LIN {X 0,Y 573.722,Z 200.489,A -85,B 0,C 180,E1 -2273.526,E2 -2273.526} C_VEL
LIN {X 0,Y 573.235,Z 198.084,A -85,B 0,C 180,E1 -2273.91,E2 -2273.91} C_VEL
LIN {X 0,Y 573.224,Z 198.082,A -85,B 0,C 180,E1 -2276.489,E2 -2276.489} C_VEL
LIN {X 0,Y 573.223,Z 198.08,A -85,B 0,C 180,E1 -2278.562,E2 -2278.562} C_VEL
LIN {X 0,Y 573.214,Z 198.078,A -85,B 0,C 180,E1 -2280.99,E2 -2280.99} C_VEL
LIN {X 0,Y 573.246,Z 198.076,A -85,B 0,C 180,E1 -2283.521,E2 -2283.521} C_VEL
LIN {X 0,Y 573.237,Z 198.083,A -85,B 0,C 180,E1 -2286.045,E2 -2286.045} C_VEL
LIN {X 0,Y 573.225,Z 198.076,A -85,B 0,C 180,E1 -2288.698,E2 -2288.698} C_VEL
LIN {X 0,Y 573.228,Z 198.081,A -85,B 0,C 180,E1 -2291.592,E2 -2291.592} C_VEL
LIN {X 0,Y 573.21,Z 198.08,A -85,B 0,C 180,E1 -2294.33,E2 -2294.33} C_VEL
LIN {X 0,Y 573.227,Z 198.079,A -85,B 0,C 180,E1 -2297.353,E2 -2297.353} C_VEL
LIN {X 0,Y 573.207,Z 198.079,A -85,B 0,C 180,E1 -2300.389,E2 -2300.389} C_VEL
LIN {X 0,Y 573.218,Z 198.079,A -85,B 0,C 180,E1 -2303.075,E2 -2303.075} C_VEL
LIN {X 0,Y 573.236,Z 198.083,A -85,B 0,C 180,E1 -2305.669,E2 -2305.669} C_VEL
LIN {X 0,Y 573.211,Z 198.079,A -85,B 0,C 180,E1 -2308.182,E2 -2308.182} C_VEL
LIN {X 0,Y 573.224,Z 198.076,A -85,B 0,C 180,E1 -2310.632,E2 -2310.632} C_VEL
LIN {X 0,Y 573.222,Z 198.086,A -85,B 0,C 180,E1 -2313.498,E2 -2313.498} C_VEL
LIN {X 0,Y 573.194,Z 198.08,A -85,B 0,C 180,E1 -2316.133,E2 -2316.133} C_VEL
LIN {X 0,Y 573.208,Z 198.079,A -85,B 0,C 180,E1 -2318.704,E2 -2318.704} C_VEL
LIN {X 0,Y 573.199,Z 198.087,A -85,B 0,C 180,E1 -2321.41,E2 -2321.41} C_VEL
LIN {X 0,Y 573.216,Z 198.081,A -85,B 0,C 180,E1 -2323.62,E2 -2323.62} C_VEL
LIN {X 0,Y 573.186,Z 198.082,A -85,B 0,C 180,E1 -2326.528,E2 -2326.528} C_VEL
LIN {X 0,Y 573.241,Z 198.079,A -85,B 0,C 180,E1 -2329.403,E2 -2329.403} C_VEL
LIN {X 0,Y 573.231,Z 198.075,A -85,B 0,C 180,E1 -2332.249,E2 -2332.249} C_VEL
LIN {X 0,Y 573.262,Z 198.081,A -85,B 0,C 180,E1 -2335.077,E2 -2335.077} C_VEL
LIN {X 0,Y 573.244,Z 198.074,A -85,B 0,C 180,E1 -2337.892,E2 -2337.892} C_VEL
LIN {X 0,Y 573.291,Z 198.074,A -85,B 0,C 180,E1 -2340.702,E2 -2340.702} C_VEL
LIN {X 0,Y 573.194,Z 198.081,A -85,B 0,C 180,E1 -2343.514,E2 -2343.514} C_VEL
LIN {X 0,Y 573.244,Z 198.074,A -85,B 0,C 180,E1 -2345.628,E2 -2345.628} C_VEL
LIN {X 0,Y 573.234,Z 198.075,A -85,B 0,C 180,E1 -2347.75,E2 -2347.75} C_VEL
LIN {X 0,Y 573.247,Z 198.081,A -85,B 0,C 180,E1 -2350.597,E2 -2350.597} C_VEL
LIN {X 0,Y 573.204,Z 198.079,A -85,B 0,C 180,E1 -2353.471,E2 -2353.471} C_VEL
LIN {X 0,Y 573.221,Z 198.082,A -85,B 0,C 180,E1 -2356.379,E2 -2356.379} C_VEL
LIN {X 0,Y 573.222,Z 198.077,A -85,B 0,C 180,E1 -2359.331,E2 -2359.331} C_VEL
LIN {X 0,Y 573.241,Z 198.081,A -85,B 0,C 180,E1 -2362.337,E2 -2362.337} C_VEL
LIN {X 0,Y 573.214,Z 198.082,A -85,B 0,C 180,E1 -2364.433,E2 -2364.433} C_VEL
LIN {X 0,Y 572.574,Z 198.165,A -85,B 0,C 180,E1 -2365.019,E2 -2365.019} C_VEL
LIN {X 0,Y 569.731,Z 198.517,A -85,B 0,C 180,E1 -2365.971,E2 -2365.971} C_VEL
LIN {X 0,Y 567.309,Z 198.818,A -85,B 0,C 180,E1 -2366.737,E2 -2366.737} C_VEL
LIN {X 0,Y 566.26,Z 198.944,A -85,B 0,C 180,E1 -2367.329,E2 -2367.329} C_VEL
LIN {X 0,Y 566.171,Z 198.955,A -85,B 0,C 180,E1 -2367.529,E2 -2367.529} C_VEL
LIN {X 0,Y 566.186,Z 198.954,A -85,B 0,C 180,E1 -2369.769,E2 -2369.769} C_VEL
LIN {X 0,Y 566.172,Z 198.962,A -85,B 0,C 180,E1 -2372.435,E2 -2372.435} C_VEL
LIN {X 0,Y 566.175,Z 198.955,A -85,B 0,C 180,E1 -2374.998,E2 -2374.998} C_VEL
LIN {X 0,Y 566.158,Z 198.957,A -85,B 0,C 180,E1 -2377.464,E2 -2377.464} C_VEL
LIN {X 0,Y 566.198,Z 198.961,A -85,B 0,C 180,E1 -2380.2,E2 -2380.2} C_VEL
LIN {X 0,Y 566.179,Z 198.954,A -85,B 0,C 180,E1 -2383.056,E2 -2383.056} C_VEL
LIN {X 0,Y 566.171,Z 198.965,A -85,B 0,C 180,E1 -2386.051,E2 -2386.051} C_VEL
LIN {X 0,Y 566.193,Z 198.952,A -85,B 0,C 180,E1 -2388.868,E2 -2388.868} C_VEL
LIN {X 0,Y 566.167,Z 198.96,A -85,B 0,C 180,E1 -2391.64,E2 -2391.64} C_VEL
LIN {X 0,Y 566.19,Z 198.956,A -85,B 0,C 180,E1 -2394.315,E2 -2394.315} C_VEL
LIN {X 0,Y 566.21,Z 198.95,A -85,B 0,C 180,E1 -2396.901,E2 -2396.901} C_VEL
LIN {X 0,Y 566.177,Z 198.958,A -85,B 0,C 180,E1 -2399.411,E2 -2399.411} C_VEL
LIN {X 0,Y 566.214,Z 198.957,A -85,B 0,C 180,E1 -2401.861,E2 -2401.861} C_VEL
LIN {X 0,Y 566.215,Z 198.951,A -85,B 0,C 180,E1 -2404.254,E2 -2404.254} C_VEL
LIN {X 0,Y 566.181,Z 198.953,A -85,B 0,C 180,E1 -2406.716,E2 -2406.716} C_VEL
LIN {X 0,Y 566.206,Z 198.959,A -85,B 0,C 180,E1 -2409.665,E2 -2409.665} C_VEL
LIN {X 0,Y 566.193,Z 198.952,A -85,B 0,C 180,E1 -2412.67,E2 -2412.67} C_VEL
LIN {X 0,Y 566.229,Z 198.955,A -85,B 0,C 180,E1 -2415.628,E2 -2415.628} C_VEL
LIN {X 0,Y 566.232,Z 198.948,A -85,B 0,C 180,E1 -2418.676,E2 -2418.676} C_VEL
LIN {X 0,Y 566.231,Z 198.956,A -85,B 0,C 180,E1 -2421.435,E2 -2421.435} C_VEL
LIN {X 0,Y 566.259,Z 198.944,A -85,B 0,C 180,E1 -2424.302,E2 -2424.302} C_VEL
LIN {X 0,Y 566.285,Z 198.942,A -85,B 0,C 180,E1 -2427.867,E2 -2427.867} C_VEL
LIN {X 0,Y 566.296,Z 198.942,A -85,B 0,C 180,E1 -2430.711,E2 -2430.711} C_VEL
LIN {X 0,Y 566.266,Z 198.948,A -85,B 0,C 180,E1 -2432.845,E2 -2432.845} C_VEL
LIN {X 0,Y 566.263,Z 198.945,A -85,B 0,C 180,E1 -2435.698,E2 -2435.698} C_VEL
LIN {X 0,Y 566.226,Z 198.951,A -85,B 0,C 180,E1 -2438.565,E2 -2438.565} C_VEL
LIN {X 0,Y 566.239,Z 198.949,A -85,B 0,C 180,E1 -2441.453,E2 -2441.453} C_VEL
LIN {X 0,Y 566.23,Z 198.951,A -85,B 0,C 180,E1 -2444.505,E2 -2444.505} C_VEL
LIN {X 0,Y 566.198,Z 198.954,A -85,B 0,C 180,E1 -2447.33,E2 -2447.33} C_VEL
LIN {X 0,Y 566.212,Z 198.952,A -85,B 0,C 180,E1 -2450.335,E2 -2450.335} C_VEL
LIN {X 0,Y 566.181,Z 198.955,A -85,B 0,C 180,E1 -2453.402,E2 -2453.402} C_VEL
LIN {X 0,Y 566.217,Z 198.95,A -85,B 0,C 180,E1 -2455.746,E2 -2455.746} C_VEL
LIN {X 0,Y 566.196,Z 198.956,A -85,B 0,C 180,E1 -2458.201,E2 -2458.201} C_VEL
LIN {X 0,Y 566.223,Z 198.955,A -85,B 0,C 180,E1 -2461.082,E2 -2461.082} C_VEL
LIN {X 0,Y 566.272,Z 199.164,A -85,B 0,C 180,E1 -2461.622,E2 -2461.622} C_VEL
LIN {X 0,Y 566.365,Z 208.652,A -85,B 0,C 180,E1 -2463.418,E2 -2463.418} C_VEL
LIN {X 0,Y 566.197,Z 222.863,A -85,B 0,C 180,E1 -2466.06,E2 -2466.06} C_VEL
LIN {X 0,Y 567.145,Z 228.431,A -85,B 0,C 180,E1 -2466.155,E2 -2466.155} C_VEL
LIN {X 0,Y 566.921,Z 329.387,A -85,B 0,C 180,E1 -2467.456,E2 -2467.456} C_VEL
LIN {X 0,Y 566.777,Z 342.831,A -85,B 0,C 180,E1 -2467.78,E2 -2467.78} C_VEL
LIN {X 0,Y 566.709,Z 354.69,A -85,B 0,C 180,E1 -2468.204,E2 -2468.204} C_VEL
LIN {X 0,Y 566.603,Z 366.89,A -85,B 0,C 180,E1 -2468.795,E2 -2468.795} C_VEL
LIN {X 0,Y 566.443,Z 377.887,A -85,B 0,C 180,E1 -2469.476,E2 -2469.476} C_VEL
LIN {X 0,Y 566.324,Z 388.435,A -85,B 0,C 180,E1 -2470.296,E2 -2470.296} C_VEL
LIN {X 0,Y 566.188,Z 398.352,A -85,B 0,C 180,E1 -2471.251,E2 -2471.251} C_VEL
LIN {X 0,Y 566.076,Z 407.08,A -85,B 0,C 180,E1 -2472.291,E2 -2472.291} C_VEL
LIN {X 0,Y 565.984,Z 415.126,A -85,B 0,C 180,E1 -2473.499,E2 -2473.499} C_VEL
LIN {X 0,Y 565.971,Z 421.457,A -85,B 0,C 180,E1 -2474.718,E2 -2474.718} C_VEL
LIN {X 0,Y 565.883,Z 426.717,A -85,B 0,C 180,E1 -2476.075,E2 -2476.075} C_VEL
LIN {X 0,Y 565.865,Z 429.598,A -85,B 0,C 180,E1 -2477.113,E2 -2477.113} C_VEL
LIN {X 0,Y 565.845,Z 431.605,A -85,B 0,C 180,E1 -2478.171,E2 -2478.171} C_VEL
LIN {X 0,Y 565.836,Z 432.73,A -85,B 0,C 180,E1 -2479.25,E2 -2479.25} C_VEL
LIN {X 0,Y 565.822,Z 432.825,A -85,B 0,C 180,E1 -2480.694,E2 -2480.694} C_VEL
LIN {X 0,Y 565.873,Z 432.026,A -85,B 0,C 180,E1 -2481.612,E2 -2481.612} C_VEL
LIN {X 0,Y 565.868,Z 430.345,A -85,B 0,C 180,E1 -2482.635,E2 -2482.635} C_VEL
LIN {X 0,Y 565.897,Z 427.33,A -85,B 0,C 180,E1 -2483.819,E2 -2483.819} C_VEL
LIN {X 0,Y 565.885,Z 422.394,A -85,B 0,C 180,E1 -2485.16,E2 -2485.16} C_VEL
LIN {X 0,Y 565.97,Z 416.825,A -85,B 0,C 180,E1 -2486.293,E2 -2486.293} C_VEL
LIN {X 0,Y 566.041,Z 409.575,A -85,B 0,C 180,E1 -2487.455,E2 -2487.455} C_VEL
LIN {X 0,Y 566.155,Z 400.734,A -85,B 0,C 180,E1 -2488.576,E2 -2488.576} C_VEL
LIN {X 0,Y 566.279,Z 391.555,A -85,B 0,C 180,E1 -2489.517,E2 -2489.517} C_VEL
LIN {X 0,Y 566.376,Z 381.392,A -85,B 0,C 180,E1 -2490.36,E2 -2490.36} C_VEL
LIN {X 0,Y 566.498,Z 370.917,A -85,B 0,C 180,E1 -2491.064,E2 -2491.064} C_VEL
LIN {X 0,Y 566.698,Z 359.05,A -85,B 0,C 180,E1 -2491.693,E2 -2491.693} C_VEL
LIN {X 0,Y 566.813,Z 346.486,A -85,B 0,C 180,E1 -2492.192,E2 -2492.192} C_VEL
LIN {X 0,Y 566.907,Z 333.732,A -85,B 0,C 180,E1 -2492.548,E2 -2492.548} C_VEL
LIN {X 0,Y 566.945,Z 319.764,A -85,B 0,C 180,E1 -2492.776,E2 -2492.776} C_VEL
LIN {X 0,Y 567.064,Z 227.64,A -85,B 0,C 180,E1 -2493.947,E2 -2493.947} C_VEL
LIN {X 0,Y 566.218,Z 222.546,A -85,B 0,C 180,E1 -2494.054,E2 -2494.054} C_VEL
LIN {X 0,Y 566.314,Z 208.588,A -85,B 0,C 180,E1 -2496.671,E2 -2496.671} C_VEL
LIN {X 0,Y 566.201,Z 198.956,A -85,B 0,C 180,E1 -2498.428,E2 -2498.428} C_VEL
LIN {X 0,Y 566.173,Z 198.962,A -85,B 0,C 180,E1 -2501.171,E2 -2501.171} C_VEL
LIN {X 0,Y 566.187,Z 198.962,A -85,B 0,C 180,E1 -2503.412,E2 -2503.412} C_VEL
LIN {X 0,Y 566.163,Z 198.958,A -85,B 0,C 180,E1 -2506.358,E2 -2506.358} C_VEL
LIN {X 0,Y 566.223,Z 198.959,A -85,B 0,C 180,E1 -2509.27,E2 -2509.27} C_VEL
LIN {X 0,Y 566.19,Z 198.953,A -85,B 0,C 180,E1 -2512.153,E2 -2512.153} C_VEL
LIN {X 0,Y 566.213,Z 198.95,A -85,B 0,C 180,E1 -2514.301,E2 -2514.301} C_VEL
LIN {X 0,Y 566.232,Z 198.957,A -85,B 0,C 180,E1 -2517.154,E2 -2517.154} C_VEL
LIN {X 0,Y 566.226,Z 198.948,A -85,B 0,C 180,E1 -2520,E2 -2520} C_VEL
LIN {X 0,Y 566.228,Z 198.955,A -85,B 0,C 180,E1 -2522.846,E2 -2522.846} C_VEL
LIN {X 0,Y 566.206,Z 198.951,A -85,B 0,C 180,E1 -2525.699,E2 -2525.699} C_VEL
LIN {X 0,Y 566.191,Z 198.957,A -85,B 0,C 180,E1 -2528.567,E2 -2528.567} C_VEL
LIN {X 0,Y 566.207,Z 198.952,A -85,B 0,C 180,E1 -2531.455,E2 -2531.455} C_VEL
LIN {X 0,Y 566.177,Z 198.959,A -85,B 0,C 180,E1 -2534.508,E2 -2534.508} C_VEL
LIN {X 0,Y 566.204,Z 198.952,A -85,B 0,C 180,E1 -2537.332,E2 -2537.332} C_VEL
LIN {X 0,Y 566.175,Z 198.959,A -85,B 0,C 180,E1 -2540.339,E2 -2540.339} C_VEL
LIN {X 0,Y 566.181,Z 198.953,A -85,B 0,C 180,E1 -2543.404,E2 -2543.404} C_VEL
LIN {X 0,Y 566.175,Z 198.955,A -85,B 0,C 180,E1 -2545.751,E2 -2545.751} C_VEL
LIN {X 0,Y 566.184,Z 198.958,A -85,B 0,C 180,E1 -2548.21,E2 -2548.21} C_VEL
LIN {X 0,Y 566.157,Z 198.958,A -85,B 0,C 180,E1 -2551.081,E2 -2551.081} C_VEL
LIN {X 0,Y 566.171,Z 198.956,A -85,B 0,C 180,E1 -2553.737,E2 -2553.737} C_VEL
LIN {X 0,Y 566.179,Z 198.961,A -85,B 0,C 180,E1 -2556.572,E2 -2556.572} C_VEL
LIN {X 0,Y 566.174,Z 198.956,A -85,B 0,C 180,E1 -2559.688,E2 -2559.688} C_VEL
LIN {X 0,Y 566.191,Z 198.959,A -85,B 0,C 180,E1 -2562.09,E2 -2562.09} C_VEL
LIN {X 0,Y 566.143,Z 198.958,A -85,B 0,C 180,E1 -2565.039,E2 -2565.039} C_VEL
LIN {X 0,Y 566.193,Z 198.961,A -85,B 0,C 180,E1 -2568.139,E2 -2568.139} C_VEL
LIN {X 0,Y 566.197,Z 198.953,A -85,B 0,C 180,E1 -2570.73,E2 -2570.73} C_VEL
LIN {X 0,Y 566.196,Z 198.958,A -85,B 0,C 180,E1 -2573.787,E2 -2573.787} C_VEL
LIN {X 0,Y 566.213,Z 198.95,A -85,B 0,C 180,E1 -2576.901,E2 -2576.901} C_VEL
LIN {X 0,Y 566.171,Z 198.958,A -85,B 0,C 180,E1 -2579.41,E2 -2579.41} C_VEL
LIN {X 0,Y 566.201,Z 198.962,A -85,B 0,C 180,E1 -2581.86,E2 -2581.86} C_VEL
LIN {X 0,Y 566.206,Z 198.956,A -85,B 0,C 180,E1 -2584.254,E2 -2584.254} C_VEL
LIN {X 0,Y 566.199,Z 198.966,A -85,B 0,C 180,E1 -2586.066,E2 -2586.066} C_VEL
LIN {X 0,Y 567.001,Z 204.188,A -85,B 0,C 180,E1 -2586.828,E2 -2586.828} C_VEL
LIN {X 0,Y 566.869,Z 223.458,A -85,B 0,C 180,E1 -2589.5,E2 -2589.5} C_VEL
LIN {X 0,Y 566.66,Z 244,A -85,B 0,C 180,E1 -2592.312,E2 -2592.312} C_VEL
LIN {X 0,Y 566.471,Z 265.283,A -85,B 0,C 180,E1 -2595.265,E2 -2595.265} C_VEL
LIN {X 0,Y 566.426,Z 270.533,A -85,B 0,C 180,E1 -2595.988,E2 -2595.988} C_VEL
LIN {X 0,Y 567.166,Z 276.627,A -85,B 0,C 180,E1 -2596.087,E2 -2596.087} C_VEL
LIN {X 0,Y 566.925,Z 379.014,A -85,B 0,C 180,E1 -2597.404,E2 -2597.404} C_VEL
LIN {X 0,Y 566.834,Z 392.262,A -85,B 0,C 180,E1 -2597.72,E2 -2597.72} C_VEL
LIN {X 0,Y 566.716,Z 404.409,A -85,B 0,C 180,E1 -2598.149,E2 -2598.149} C_VEL
LIN {X 0,Y 566.626,Z 416.087,A -85,B 0,C 180,E1 -2598.705,E2 -2598.705} C_VEL
LIN {X 0,Y 566.485,Z 426.922,A -85,B 0,C 180,E1 -2599.367,E2 -2599.367} C_VEL
LIN {X 0,Y 566.337,Z 437.551,A -85,B 0,C 180,E1 -2600.176,E2 -2600.176} C_VEL
LIN {X 0,Y 566.206,Z 447.122,A -85,B 0,C 180,E1 -2601.075,E2 -2601.075} C_VEL
LIN {X 0,Y 566.112,Z 454.967,A -85,B 0,C 180,E1 -2601.972,E2 -2601.972} C_VEL
LIN {X 0,Y 566,Z 462.627,A -85,B 0,C 180,E1 -2603.047,E2 -2603.047} C_VEL
LIN {X 0,Y 566.004,Z 469.683,A -85,B 0,C 180,E1 -2604.3,E2 -2604.3} C_VEL
LIN {X 0,Y 565.933,Z 474.374,A -85,B 0,C 180,E1 -2605.371,E2 -2605.371} C_VEL
LIN {X 0,Y 565.927,Z 477.959,A -85,B 0,C 180,E1 -2606.44,E2 -2606.44} C_VEL
LIN {X 0,Y 565.878,Z 479.808,A -85,B 0,C 180,E1 -2607.153,E2 -2607.153} C_VEL
LIN {X 0,Y 565.846,Z 482.184,A -85,B 0,C 180,E1 -2608.577,E2 -2608.577} C_VEL
LIN {X 0,Y 565.839,Z 483,A -85,B 0,C 180,E1 -2610,E2 -2610} C_VEL
LIN {X 0,Y 565.846,Z 482.186,A -85,B 0,C 180,E1 -2611.423,E2 -2611.423} C_VEL
LIN {X 0,Y 565.878,Z 479.811,A -85,B 0,C 180,E1 -2612.847,E2 -2612.847} C_VEL
LIN {X 0,Y 565.926,Z 476.897,A -85,B 0,C 180,E1 -2613.916,E2 -2613.916} C_VEL
LIN {X 0,Y 565.878,Z 472.951,A -85,B 0,C 180,E1 -2614.987,E2 -2614.987} C_VEL
LIN {X 0,Y 566.004,Z 467.871,A -85,B 0,C 180,E1 -2616.058,E2 -2616.058} C_VEL
LIN {X 0,Y 566.04,Z 461.473,A -85,B 0,C 180,E1 -2617.131,E2 -2617.131} C_VEL
LIN {X 0,Y 566.133,Z 453.486,A -85,B 0,C 180,E1 -2618.207,E2 -2618.207} C_VEL
LIN {X 0,Y 566.228,Z 445.345,A -85,B 0,C 180,E1 -2619.104,E2 -2619.104} C_VEL
LIN {X 0,Y 566.35,Z 435.413,A -85,B 0,C 180,E1 -2620.004,E2 -2620.004} C_VEL
LIN {X 0,Y 566.508,Z 424.305,A -85,B 0,C 180,E1 -2620.807,E2 -2620.807} C_VEL
LIN {X 0,Y 566.658,Z 413.2,A -85,B 0,C 180,E1 -2621.444,E2 -2621.444} C_VEL
LIN {X 0,Y 566.757,Z 401.015,A -85,B 0,C 180,E1 -2621.986,E2 -2621.986} C_VEL
LIN {X 0,Y 566.895,Z 388.233,A -85,B 0,C 180,E1 -2622.392,E2 -2622.392} C_VEL
LIN {X 0,Y 566.972,Z 374.699,A -85,B 0,C 180,E1 -2622.663,E2 -2622.663} C_VEL
LIN {X 0,Y 567.064,Z 275.054,A -85,B 0,C 180,E1 -2623.935,E2 -2623.935} C_VEL
LIN {X 0,Y 566.423,Z 270.451,A -85,B 0,C 180,E1 -2624.023,E2 -2624.023} C_VEL
LIN {X 0,Y 566.643,Z 248.046,A -85,B 0,C 180,E1 -2627.125,E2 -2627.125} C_VEL
LIN {X 0,Y 566.893,Z 226.441,A -85,B 0,C 180,E1 -2630.12,E2 -2630.12} C_VEL
LIN {X 0,Y 567.128,Z 206.124,A -85,B 0,C 180,E1 -2632.974,E2 -2632.974} C_VEL
LIN {X 0,Y 566.842,Z 202.208,A -85,B 0,C 180,E1 -2633.547,E2 -2633.547} C_VEL
LIN {X 0,Y 566.214,Z 198.959,A -85,B 0,C 180,E1 -2634.08,E2 -2634.08} C_VEL
LIN {X 0,Y 566.19,Z 198.956,A -85,B 0,C 180,E1 -2636.655,E2 -2636.655} C_VEL
LIN {X 0,Y 566.179,Z 198.955,A -85,B 0,C 180,E1 -2638.95,E2 -2638.95} C_VEL
LIN {X 0,Y 566.179,Z 198.956,A -85,B 0,C 180,E1 -2641.419,E2 -2641.419} C_VEL
LIN {X 0,Y 566.193,Z 198.961,A -85,B 0,C 180,E1 -2643.953,E2 -2643.953} C_VEL
LIN {X 0,Y 566.194,Z 198.953,A -85,B 0,C 180,E1 -2646.566,E2 -2646.566} C_VEL
LIN {X 0,Y 566.189,Z 198.959,A -85,B 0,C 180,E1 -2649.682,E2 -2649.682} C_VEL
LIN {X 0,Y 566.187,Z 198.959,A -85,B 0,C 180,E1 -2652.084,E2 -2652.084} C_VEL
LIN {X 0,Y 566.143,Z 198.959,A -85,B 0,C 180,E1 -2655.032,E2 -2655.032} C_VEL
LIN {X 0,Y 566.193,Z 198.959,A -85,B 0,C 180,E1 -2657.91,E2 -2657.91} C_VEL
LIN {X 0,Y 566.181,Z 198.953,A -85,B 0,C 180,E1 -2660.723,E2 -2660.723} C_VEL
LIN {X 0,Y 566.179,Z 198.961,A -85,B 0,C 180,E1 -2663.78,E2 -2663.78} C_VEL
LIN {X 0,Y 566.188,Z 198.953,A -85,B 0,C 180,E1 -2666.26,E2 -2666.26} C_VEL
LIN {X 0,Y 566.157,Z 198.958,A -85,B 0,C 180,E1 -2668.919,E2 -2668.919} C_VEL
LIN {X 0,Y 566.182,Z 198.957,A -85,B 0,C 180,E1 -2671.855,E2 -2671.855} C_VEL
LIN {X 0,Y 566.175,Z 198.954,A -85,B 0,C 180,E1 -2674.249,E2 -2674.249} C_VEL
LIN {X 0,Y 566.154,Z 198.967,A -85,B 0,C 180,E1 -2677.367,E2 -2677.367} C_VEL
LIN {X 0,Y 566.175,Z 198.959,A -85,B 0,C 180,E1 -2679.661,E2 -2679.661} C_VEL
LIN {X 0,Y 566.221,Z 198.952,A -85,B 0,C 180,E1 -2682.867,E2 -2682.867} C_VEL
LIN {X 0,Y 566.176,Z 198.958,A -85,B 0,C 180,E1 -2685.625,E2 -2685.625} C_VEL
LIN {X 0,Y 566.236,Z 198.949,A -85,B 0,C 180,E1 -2688.643,E2 -2688.643} C_VEL
LIN {X 0,Y 566.191,Z 198.957,A -85,B 0,C 180,E1 -2691.433,E2 -2691.433} C_VEL
LIN {X 0,Y 566.205,Z 198.951,A -85,B 0,C 180,E1 -2694.301,E2 -2694.301} C_VEL
LIN {X 0,Y 566.227,Z 198.955,A -85,B 0,C 180,E1 -2697.154,E2 -2697.154} C_VEL
LIN {X 0,Y 566.225,Z 198.948,A -85,B 0,C 180,E1 -2700,E2 -2700} C_VEL
LIN {X 0,Y 566.231,Z 198.957,A -85,B 0,C 180,E1 -2702.846,E2 -2702.846} C_VEL
LIN {X 0,Y 566.212,Z 198.95,A -85,B 0,C 180,E1 -2705.699,E2 -2705.699} C_VEL
LIN {X 0,Y 566.189,Z 198.952,A -85,B 0,C 180,E1 -2707.847,E2 -2707.847} C_VEL
LIN {X 0,Y 566.222,Z 198.958,A -85,B 0,C 180,E1 -2710.73,E2 -2710.73} C_VEL
LIN {X 0,Y 566.162,Z 198.956,A -85,B 0,C 180,E1 -2713.642,E2 -2713.642} C_VEL
LIN {X 0,Y 566.185,Z 198.963,A -85,B 0,C 180,E1 -2716.588,E2 -2716.588} C_VEL
LIN {X 0,Y 566.165,Z 198.955,A -85,B 0,C 180,E1 -2719.582,E2 -2719.582} C_VEL
LIN {X 0,Y 566.197,Z 198.953,A -85,B 0,C 180,E1 -2721.862,E2 -2721.862} C_VEL
LIN {X 0,Y 566.162,Z 198.959,A -85,B 0,C 180,E1 -2724.433,E2 -2724.433} C_VEL
LIN {X 0,Y 566.182,Z 198.953,A -85,B 0,C 180,E1 -2727.34,E2 -2727.34} C_VEL
LIN {X 0,Y 566.171,Z 198.955,A -85,B 0,C 180,E1 -2727.529,E2 -2727.529} C_VEL
LIN {X 0,Y 565.493,Z 199.046,A -85,B 0,C 180,E1 -2728.123,E2 -2728.123} C_VEL
LIN {X 0,Y 562.627,Z 199.401,A -85,B 0,C 180,E1 -2729.087,E2 -2729.087} C_VEL
LIN {X 0,Y 560.217,Z 199.701,A -85,B 0,C 180,E1 -2729.862,E2 -2729.862} C_VEL
LIN {X 0,Y 559.19,Z 199.832,A -85,B 0,C 180,E1 -2730.461,E2 -2730.461} C_VEL
LIN {X 0,Y 559.111,Z 199.836,A -85,B 0,C 180,E1 -2730.664,E2 -2730.664} C_VEL
LIN {X 0,Y 559.136,Z 199.832,A -85,B 0,C 180,E1 -2733.576,E2 -2733.576} C_VEL
LIN {X 0,Y 559.15,Z 199.835,A -85,B 0,C 180,E1 -2736.454,E2 -2736.454} C_VEL
LIN {X 0,Y 559.159,Z 199.833,A -85,B 0,C 180,E1 -2739.867,E2 -2739.867} C_VEL
LIN {X 0,Y 559.139,Z 199.832,A -85,B 0,C 180,E1 -2742.745,E2 -2742.745} C_VEL
LIN {X 0,Y 559.123,Z 199.838,A -85,B 0,C 180,E1 -2745.764,E2 -2745.764} C_VEL
LIN {X 0,Y 559.169,Z 199.833,A -85,B 0,C 180,E1 -2748.236,E2 -2748.236} C_VEL
LIN {X 0,Y 559.154,Z 199.829,A -85,B 0,C 180,E1 -2751.194,E2 -2751.194} C_VEL
LIN {X 0,Y 559.15,Z 199.837,A -85,B 0,C 180,E1 -2753.795,E2 -2753.795} C_VEL
LIN {X 0,Y 559.158,Z 199.83,A -85,B 0,C 180,E1 -2756.429,E2 -2756.429} C_VEL
LIN {X 0,Y 559.149,Z 199.83,A -85,B 0,C 180,E1 -2758.984,E2 -2758.984} C_VEL
LIN {X 0,Y 559.155,Z 199.836,A -85,B 0,C 180,E1 -2761.621,E2 -2761.621} C_VEL
LIN {X 0,Y 559.187,Z 199.831,A -85,B 0,C 180,E1 -2763.906,E2 -2763.906} C_VEL
LIN {X 0,Y 559.146,Z 199.83,A -85,B 0,C 180,E1 -2766.57,E2 -2766.57} C_VEL
LIN {X 0,Y 559.172,Z 199.833,A -85,B 0,C 180,E1 -2769.398,E2 -2769.398} C_VEL
LIN {X 0,Y 559.138,Z 199.838,A -85,B 0,C 180,E1 -2771.688,E2 -2771.688} C_VEL
LIN {X 0,Y 559.161,Z 199.831,A -85,B 0,C 180,E1 -2773.95,E2 -2773.95} C_VEL
LIN {X 0,Y 559.167,Z 199.828,A -85,B 0,C 180,E1 -2776.186,E2 -2776.186} C_VEL
LIN {X 0,Y 559.193,Z 199.829,A -85,B 0,C 180,E1 -2779.135,E2 -2779.135} C_VEL
LIN {X 0,Y 559.199,Z 199.824,A -85,B 0,C 180,E1 -2782.055,E2 -2782.055} C_VEL
LIN {X 0,Y 559.253,Z 199.821,A -85,B 0,C 180,E1 -2784.954,E2 -2784.954} C_VEL
LIN {X 0,Y 559.256,Z 199.818,A -85,B 0,C 180,E1 -2787.84,E2 -2787.84} C_VEL
LIN {X 0,Y 559.267,Z 199.817,A -85,B 0,C 180,E1 -2790.72,E2 -2790.72} C_VEL
LIN {X 0,Y 559.234,Z 199.824,A -85,B 0,C 180,E1 -2792.881,E2 -2792.881} C_VEL
LIN {X 0,Y 559.231,Z 199.82,A -85,B 0,C 180,E1 -2795.77,E2 -2795.77} C_VEL
LIN {X 0,Y 559.185,Z 199.829,A -85,B 0,C 180,E1 -2798.674,E2 -2798.674} C_VEL
LIN {X 0,Y 559.202,Z 199.824,A -85,B 0,C 180,E1 -2801.599,E2 -2801.599} C_VEL
LIN {X 0,Y 559.195,Z 199.828,A -85,B 0,C 180,E1 -2804.594,E2 -2804.594} C_VEL
LIN {X 0,Y 559.157,Z 199.829,A -85,B 0,C 180,E1 -2807.555,E2 -2807.555} C_VEL
LIN {X 0,Y 559.178,Z 199.832,A -85,B 0,C 180,E1 -2810.602,E2 -2810.602} C_VEL
LIN {X 0,Y 559.137,Z 199.831,A -85,B 0,C 180,E1 -2813.714,E2 -2813.714} C_VEL
LIN {X 0,Y 559.19,Z 199.827,A -85,B 0,C 180,E1 -2816.094,E2 -2816.094} C_VEL
LIN {X 0,Y 559.154,Z 199.838,A -85,B 0,C 180,E1 -2818.527,E2 -2818.527} C_VEL
LIN {X 0,Y 559.231,Z 199.938,A -85,B 0,C 180,E1 -2821.532,E2 -2821.532} C_VEL
LIN {X 0,Y 559.348,Z 208.336,A -85,B 0,C 180,E1 -2823.127,E2 -2823.127} C_VEL
LIN {X 0,Y 559.155,Z 222.71,A -85,B 0,C 180,E1 -2825.871,E2 -2825.871} C_VEL
LIN {X 0,Y 560.287,Z 230.608,A -85,B 0,C 180,E1 -2826.009,E2 -2826.009} C_VEL
LIN {X 0,Y 560.005,Z 328.988,A -85,B 0,C 180,E1 -2827.291,E2 -2827.291} C_VEL
LIN {X 0,Y 559.828,Z 342.195,A -85,B 0,C 180,E1 -2827.606,E2 -2827.606} C_VEL
LIN {X 0,Y 559.787,Z 353.765,A -85,B 0,C 180,E1 -2828.017,E2 -2828.017} C_VEL
LIN {X 0,Y 559.639,Z 365.973,A -85,B 0,C 180,E1 -2828.602,E2 -2828.602} C_VEL
LIN {X 0,Y 559.455,Z 376.579,A -85,B 0,C 180,E1 -2829.254,E2 -2829.254} C_VEL
LIN {X 0,Y 559.291,Z 385.919,A -85,B 0,C 180,E1 -2829.958,E2 -2829.958} C_VEL
LIN {X 0,Y 559.181,Z 395.174,A -85,B 0,C 180,E1 -2830.805,E2 -2830.805} C_VEL
LIN {X 0,Y 559.071,Z 403.824,A -85,B 0,C 180,E1 -2831.773,E2 -2831.773} C_VEL
LIN {X 0,Y 558.911,Z 412.404,A -85,B 0,C 180,E1 -2832.967,E2 -2832.967} C_VEL
LIN {X 0,Y 558.875,Z 419.383,A -85,B 0,C 180,E1 -2834.21,E2 -2834.21} C_VEL
LIN {X 0,Y 558.822,Z 425.053,A -85,B 0,C 180,E1 -2835.536,E2 -2835.536} C_VEL
LIN {X 0,Y 558.778,Z 429.025,A -85,B 0,C 180,E1 -2836.837,E2 -2836.837} C_VEL
LIN {X 0,Y 558.748,Z 431.673,A -85,B 0,C 180,E1 -2838.192,E2 -2838.192} C_VEL
LIN {X 0,Y 558.748,Z 432.673,A -85,B 0,C 180,E1 -2839.152,E2 -2839.152} C_VEL
LIN {X 0,Y 558.765,Z 432.994,A -85,B 0,C 180,E1 -2840.099,E2 -2840.099} C_VEL
LIN {X 0,Y 558.738,Z 432.449,A -85,B 0,C 180,E1 -2841.24,E2 -2841.24} C_VEL
LIN {X 0,Y 558.768,Z 430.863,A -85,B 0,C 180,E1 -2842.401,E2 -2842.401} C_VEL
LIN {X 0,Y 558.822,Z 427.625,A -85,B 0,C 180,E1 -2843.766,E2 -2843.766} C_VEL
LIN {X 0,Y 558.821,Z 424.027,A -85,B 0,C 180,E1 -2844.824,E2 -2844.824} C_VEL
LIN {X 0,Y 558.854,Z 418.345,A -85,B 0,C 180,E1 -2846.089,E2 -2846.089} C_VEL
LIN {X 0,Y 558.956,Z 411.426,A -85,B 0,C 180,E1 -2847.272,E2 -2847.272} C_VEL
LIN {X 0,Y 559.06,Z 404.013,A -85,B 0,C 180,E1 -2848.293,E2 -2848.293} C_VEL
LIN {X 0,Y 559.196,Z 395.041,A -85,B 0,C 180,E1 -2849.298,E2 -2849.298} C_VEL
LIN {X 0,Y 559.322,Z 385.446,A -85,B 0,C 180,E1 -2850.17,E2 -2850.17} C_VEL
LIN {X 0,Y 559.47,Z 374.558,A -85,B 0,C 180,E1 -2850.975,E2 -2850.975} C_VEL
LIN {X 0,Y 559.658,Z 362.871,A -85,B 0,C 180,E1 -2851.652,E2 -2851.652} C_VEL
LIN {X 0,Y 559.809,Z 350.028,A -85,B 0,C 180,E1 -2852.22,E2 -2852.22} C_VEL
LIN {X 0,Y 559.966,Z 337.46,A -85,B 0,C 180,E1 -2852.614,E2 -2852.614} C_VEL
LIN {X 0,Y 560.059,Z 323.509,A -85,B 0,C 180,E1 -2852.886,E2 -2852.886} C_VEL
LIN {X 0,Y 560.235,Z 228.764,A -85,B 0,C 180,E1 -2854.106,E2 -2854.106} C_VEL
LIN {X 0,Y 559.2,Z 222.638,A -85,B 0,C 180,E1 -2854.229,E2 -2854.229} C_VEL
LIN {X 0,Y 559.271,Z 208.735,A -85,B 0,C 180,E1 -2856.801,E2 -2856.801} C_VEL
LIN {X 0,Y 559.161,Z 199.833,A -85,B 0,C 180,E1 -2858.393,E2 -2858.393} C_VEL
LIN {X 0,Y 559.125,Z 199.837,A -85,B 0,C 180,E1 -2860.925,E2 -2860.925} C_VEL
LIN {X 0,Y 559.161,Z 199.836,A -85,B 0,C 180,E1 -2863.197,E2 -2863.197} C_VEL
LIN {X 0,Y 559.133,Z 199.834,A -85,B 0,C 180,E1 -2866.183,E2 -2866.183} C_VEL
LIN {X 0,Y 559.203,Z 199.832,A -85,B 0,C 180,E1 -2869.134,E2 -2869.134} C_VEL
LIN {X 0,Y 559.158,Z 199.83,A -85,B 0,C 180,E1 -2872.053,E2 -2872.053} C_VEL
LIN {X 0,Y 559.212,Z 199.828,A -85,B 0,C 180,E1 -2874.953,E2 -2874.953} C_VEL
LIN {X 0,Y 559.192,Z 199.826,A -85,B 0,C 180,E1 -2877.839,E2 -2877.839} C_VEL
LIN {X 0,Y 559.226,Z 199.825,A -85,B 0,C 180,E1 -2880.72,E2 -2880.72} C_VEL
LIN {X 0,Y 559.193,Z 199.832,A -85,B 0,C 180,E1 -2882.882,E2 -2882.882} C_VEL
LIN {X 0,Y 559.174,Z 199.826,A -85,B 0,C 180,E1 -2885.771,E2 -2885.771} C_VEL
LIN {X 0,Y 559.147,Z 199.836,A -85,B 0,C 180,E1 -2888.675,E2 -2888.675} C_VEL
LIN {X 0,Y 559.159,Z 199.829,A -85,B 0,C 180,E1 -2891.602,E2 -2891.602} C_VEL
LIN {X 0,Y 559.145,Z 199.836,A -85,B 0,C 180,E1 -2894.597,E2 -2894.597} C_VEL
LIN {X 0,Y 559.159,Z 199.828,A -85,B 0,C 180,E1 -2897.557,E2 -2897.557} C_VEL
LIN {X 0,Y 559.14,Z 199.839,A -85,B 0,C 180,E1 -2900.606,E2 -2900.606} C_VEL
LIN {X 0,Y 559.118,Z 199.833,A -85,B 0,C 180,E1 -2903.718,E2 -2903.718} C_VEL
LIN {X 0,Y 559.15,Z 199.832,A -85,B 0,C 180,E1 -2906.099,E2 -2906.099} C_VEL
LIN {X 0,Y 559.13,Z 199.841,A -85,B 0,C 180,E1 -2908.532,E2 -2908.532} C_VEL
LIN {X 0,Y 559.112,Z 199.835,A -85,B 0,C 180,E1 -2911.278,E2 -2911.278} C_VEL
LIN {X 0,Y 559.127,Z 199.835,A -85,B 0,C 180,E1 -2913.952,E2 -2913.952} C_VEL
LIN {X 0,Y 559.153,Z 199.838,A -85,B 0,C 180,E1 -2916.455,E2 -2916.455} C_VEL
LIN {X 0,Y 559.14,Z 199.833,A -85,B 0,C 180,E1 -2918.937,E2 -2918.937} C_VEL
LIN {X 0,Y 559.159,Z 199.831,A -85,B 0,C 180,E1 -2921.771,E2 -2921.771} C_VEL
LIN {X 0,Y 559.11,Z 199.836,A -85,B 0,C 180,E1 -2924.743,E2 -2924.743} C_VEL
LIN {X 0,Y 559.136,Z 199.831,A -85,B 0,C 180,E1 -2927.26,E2 -2927.26} C_VEL
LIN {X 0,Y 559.158,Z 199.838,A -85,B 0,C 180,E1 -2930.138,E2 -2930.138} C_VEL
LIN {X 0,Y 559.126,Z 199.833,A -85,B 0,C 180,E1 -2932.895,E2 -2932.895} C_VEL
LIN {X 0,Y 559.149,Z 199.839,A -85,B 0,C 180,E1 -2936.054,E2 -2936.054} C_VEL
LIN {X 0,Y 559.144,Z 199.831,A -85,B 0,C 180,E1 -2938.984,E2 -2938.984} C_VEL
LIN {X 0,Y 559.157,Z 199.836,A -85,B 0,C 180,E1 -2941.622,E2 -2941.622} C_VEL
LIN {X 0,Y 559.168,Z 199.829,A -85,B 0,C 180,E1 -2944.704,E2 -2944.704} C_VEL
LIN {X 0,Y 559.168,Z 199.868,A -85,B 0,C 180,E1 -2945.943,E2 -2945.943} C_VEL
LIN {X 0,Y 560.049,Z 205.262,A -85,B 0,C 180,E1 -2946.74,E2 -2946.74} C_VEL
LIN {X 0,Y 559.875,Z 224.341,A -85,B 0,C 180,E1 -2949.425,E2 -2949.425} C_VEL
LIN {X 0,Y 559.613,Z 246.236,A -85,B 0,C 180,E1 -2952.46,E2 -2952.46} C_VEL
LIN {X 0,Y 559.456,Z 265.298,A -85,B 0,C 180,E1 -2955.079,E2 -2955.079} C_VEL
LIN {X 0,Y 559.425,Z 270.533,A -85,B 0,C 180,E1 -2955.81,E2 -2955.81} C_VEL
LIN {X 0,Y 560.282,Z 277.358,A -85,B 0,C 180,E1 -2955.922,E2 -2955.922} C_VEL
LIN {X 0,Y 560.007,Z 379.014,A -85,B 0,C 180,E1 -2957.245,E2 -2957.245} C_VEL
LIN {X 0,Y 559.895,Z 392.261,A -85,B 0,C 180,E1 -2957.565,E2 -2957.565} C_VEL
LIN {X 0,Y 559.753,Z 404.409,A -85,B 0,C 180,E1 -2957.999,E2 -2957.999} C_VEL
LIN {X 0,Y 559.667,Z 415.834,A -85,B 0,C 180,E1 -2958.548,E2 -2958.548} C_VEL
LIN {X 0,Y 559.503,Z 426.92,A -85,B 0,C 180,E1 -2959.232,E2 -2959.232} C_VEL
LIN {X 0,Y 559.317,Z 437.549,A -85,B 0,C 180,E1 -2960.052,E2 -2960.052} C_VEL
LIN {X 0,Y 559.161,Z 447.122,A -85,B 0,C 180,E1 -2960.962,E2 -2960.962} C_VEL
LIN {X 0,Y 559.049,Z 454.967,A -85,B 0,C 180,E1 -2961.87,E2 -2961.87} C_VEL
LIN {X 0,Y 558.942,Z 462.627,A -85,B 0,C 180,E1 -2962.959,E2 -2962.959} C_VEL
LIN {X 0,Y 558.935,Z 469.682,A -85,B 0,C 180,E1 -2964.227,E2 -2964.227} C_VEL
LIN {X 0,Y 558.826,Z 474.375,A -85,B 0,C 180,E1 -2965.312,E2 -2965.312} C_VEL
LIN {X 0,Y 558.836,Z 477.959,A -85,B 0,C 180,E1 -2966.395,E2 -2966.395} C_VEL
LIN {X 0,Y 558.799,Z 479.808,A -85,B 0,C 180,E1 -2967.117,E2 -2967.117} C_VEL
LIN {X 0,Y 558.745,Z 482.184,A -85,B 0,C 180,E1 -2968.559,E2 -2968.559} C_VEL
LIN {X 0,Y 558.74,Z 483,A -85,B 0,C 180,E1 -2970,E2 -2970} C_VEL
LIN {X 0,Y 558.745,Z 482.185,A -85,B 0,C 180,E1 -2971.441,E2 -2971.441} C_VEL
LIN {X 0,Y 558.799,Z 479.811,A -85,B 0,C 180,E1 -2972.883,E2 -2972.883} C_VEL
LIN {X 0,Y 558.844,Z 476.897,A -85,B 0,C 180,E1 -2973.966,E2 -2973.966} C_VEL
LIN {X 0,Y 558.798,Z 472.951,A -85,B 0,C 180,E1 -2975.05,E2 -2975.05} C_VEL
LIN {X 0,Y 558.92,Z 467.871,A -85,B 0,C 180,E1 -2976.135,E2 -2976.135} C_VEL
LIN {X 0,Y 558.977,Z 461.473,A -85,B 0,C 180,E1 -2977.222,E2 -2977.222} C_VEL
LIN {X 0,Y 559.098,Z 453.485,A -85,B 0,C 180,E1 -2978.311,E2 -2978.311} C_VEL
LIN {X 0,Y 559.184,Z 445.344,A -85,B 0,C 180,E1 -2979.22,E2 -2979.22} C_VEL
LIN {X 0,Y 559.36,Z 435.412,A -85,B 0,C 180,E1 -2980.13,E2 -2980.13} C_VEL
LIN {X 0,Y 559.51,Z 424.383,A -85,B 0,C 180,E1 -2980.938,E2 -2980.938} C_VEL
LIN {X 0,Y 559.701,Z 412.165,A -85,B 0,C 180,E1 -2981.642,E2 -2981.642} C_VEL
LIN {X 0,Y 559.829,Z 399.808,A -85,B 0,C 180,E1 -2982.183,E2 -2982.183} C_VEL
LIN {X 0,Y 559.988,Z 387.318,A -85,B 0,C 180,E1 -2982.571,E2 -2982.571} C_VEL
LIN {X 0,Y 560.056,Z 374.698,A -85,B 0,C 180,E1 -2982.822,E2 -2982.822} C_VEL
LIN {X 0,Y 560.228,Z 276.312,A -85,B 0,C 180,E1 -2984.093,E2 -2984.093} C_VEL
LIN {X 0,Y 559.431,Z 270.451,A -85,B 0,C 180,E1 -2984.202,E2 -2984.202} C_VEL
LIN {X 0,Y 559.626,Z 247.706,A -85,B 0,C 180,E1 -2987.362,E2 -2987.362} C_VEL
LIN {X 0,Y 559.904,Z 226.166,A -85,B 0,C 180,E1 -2990.382,E2 -2990.382} C_VEL
LIN {X 0,Y 560.175,Z 205.954,A -85,B 0,C 180,E1 -2993.264,E2 -2993.264} C_VEL
LIN {X 0,Y 559.17,Z 199.836,A -85,B 0,C 180,E1 -2994.205,E2 -2994.205} C_VEL
LIN {X 0,Y 559.154,Z 199.831,A -85,B 0,C 180,E1 -2996.9,E2 -2996.9} C_VEL
LIN {X 0,Y 559.137,Z 199.838,A -85,B 0,C 180,E1 -2999.855,E2 -2999.855} C_VEL
LIN {X 0,Y 559.143,Z 199.831,A -85,B 0,C 180,E1 -3002.712,E2 -3002.712} C_VEL
LIN {X 0,Y 559.129,Z 199.833,A -85,B 0,C 180,E1 -3005.319,E2 -3005.319} C_VEL
LIN {X 0,Y 559.113,Z 199.842,A -85,B 0,C 180,E1 -3008.014,E2 -3008.014} C_VEL
LIN {X 0,Y 559.166,Z 199.828,A -85,B 0,C 180,E1 -3011.051,E2 -3011.051} C_VEL
LIN {X 0,Y 559.134,Z 199.84,A -85,B 0,C 180,E1 -3013.728,E2 -3013.728} C_VEL
LIN {X 0,Y 559.14,Z 199.831,A -85,B 0,C 180,E1 -3016.797,E2 -3016.797} C_VEL
LIN {X 0,Y 559.142,Z 199.832,A -85,B 0,C 180,E1 -3019.186,E2 -3019.186} C_VEL
LIN {X 0,Y 559.097,Z 199.841,A -85,B 0,C 180,E1 -3021.979,E2 -3021.979} C_VEL
LIN {X 0,Y 559.119,Z 199.833,A -85,B 0,C 180,E1 -3024.675,E2 -3024.675} C_VEL
LIN {X 0,Y 559.135,Z 199.838,A -85,B 0,C 180,E1 -3027.358,E2 -3027.358} C_VEL
LIN {X 0,Y 559.106,Z 199.836,A -85,B 0,C 180,E1 -3030.139,E2 -3030.139} C_VEL
LIN {X 0,Y 559.149,Z 199.83,A -85,B 0,C 180,E1 -3032.286,E2 -3032.286} C_VEL
LIN {X 0,Y 559.131,Z 199.833,A -85,B 0,C 180,E1 -3034.81,E2 -3034.81} C_VEL
LIN {X 0,Y 559.113,Z 199.839,A -85,B 0,C 180,E1 -3037.066,E2 -3037.066} C_VEL
LIN {X 0,Y 559.139,Z 199.839,A -85,B 0,C 180,E1 -3039.394,E2 -3039.394} C_VEL
LIN {X 0,Y 559.158,Z 199.829,A -85,B 0,C 180,E1 -3042.443,E2 -3042.443} C_VEL
LIN {X 0,Y 559.14,Z 199.837,A -85,B 0,C 180,E1 -3045.44,E2 -3045.44} C_VEL
LIN {X 0,Y 559.18,Z 199.827,A -85,B 0,C 180,E1 -3048.587,E2 -3048.587} C_VEL
LIN {X 0,Y 559.146,Z 199.836,A -85,B 0,C 180,E1 -3051.325,E2 -3051.325} C_VEL
LIN {X 0,Y 559.173,Z 199.827,A -85,B 0,C 180,E1 -3054.229,E2 -3054.229} C_VEL
LIN {X 0,Y 559.192,Z 199.832,A -85,B 0,C 180,E1 -3057.118,E2 -3057.118} C_VEL
LIN {X 0,Y 559.196,Z 199.824,A -85,B 0,C 180,E1 -3060,E2 -3060} C_VEL
LIN {X 0,Y 559.196,Z 199.834,A -85,B 0,C 180,E1 -3062.881,E2 -3062.881} C_VEL
LIN {X 0,Y 559.182,Z 199.825,A -85,B 0,C 180,E1 -3065.77,E2 -3065.77} C_VEL
LIN {X 0,Y 559.157,Z 199.829,A -85,B 0,C 180,E1 -3067.947,E2 -3067.947} C_VEL
LIN {X 0,Y 559.201,Z 199.83,A -85,B 0,C 180,E1 -3070.866,E2 -3070.866} C_VEL
LIN {X 0,Y 559.132,Z 199.832,A -85,B 0,C 180,E1 -3073.817,E2 -3073.817} C_VEL
LIN {X 0,Y 559.159,Z 199.835,A -85,B 0,C 180,E1 -3076.803,E2 -3076.803} C_VEL
LIN {X 0,Y 559.128,Z 199.833,A -85,B 0,C 180,E1 -3079.839,E2 -3079.839} C_VEL
LIN {X 0,Y 559.14,Z 199.835,A -85,B 0,C 180,E1 -3082.153,E2 -3082.153} C_VEL
LIN {X 0,Y 559.155,Z 199.829,A -85,B 0,C 180,E1 -3085.195,E2 -3085.195} C_VEL
LIN {X 0,Y 559.149,Z 199.83,A -85,B 0,C 180,E1 -3087.714,E2 -3087.714} C_VEL
LIN {X 0,Y 559.111,Z 199.836,A -85,B 0,C 180,E1 -3090.664,E2 -3090.664} C_VEL
LIN {X 0,Y 558.45,Z 199.919,A -85,B 0,C 180,E1 -3091.266,E2 -3091.266} C_VEL
LIN {X 0,Y 555.586,Z 200.282,A -85,B 0,C 180,E1 -3092.242,E2 -3092.242} C_VEL
LIN {X 0,Y 553.174,Z 200.577,A -85,B 0,C 180,E1 -3093.028,E2 -3093.028} C_VEL
LIN {X 0,Y 552.157,Z 200.702,A -85,B 0,C 180,E1 -3093.634,E2 -3093.634} C_VEL
LIN {X 0,Y 552.084,Z 200.713,A -85,B 0,C 180,E1 -3093.84,E2 -3093.84} C_VEL
LIN {X 0,Y 552.078,Z 200.713,A -85,B 0,C 180,E1 -3096.749,E2 -3096.749} C_VEL
LIN {X 0,Y 552.12,Z 200.706,A -85,B 0,C 180,E1 -3099.528,E2 -3099.528} C_VEL
LIN {X 0,Y 552.098,Z 200.713,A -85,B 0,C 180,E1 -3102.419,E2 -3102.419} C_VEL
LIN {X 0,Y 552.067,Z 200.714,A -85,B 0,C 180,E1 -3105.566,E2 -3105.566} C_VEL
LIN {X 0,Y 552.117,Z 200.706,A -85,B 0,C 180,E1 -3108.679,E2 -3108.679} C_VEL
LIN {X 0,Y 552.096,Z 200.71,A -85,B 0,C 180,E1 -3111.414,E2 -3111.414} C_VEL
LIN {X 0,Y 552.091,Z 200.714,A -85,B 0,C 180,E1 -3114.161,E2 -3114.161} C_VEL
LIN {X 0,Y 552.11,Z 200.706,A -85,B 0,C 180,E1 -3116.818,E2 -3116.818} C_VEL
LIN {X 0,Y 552.097,Z 200.711,A -85,B 0,C 180,E1 -3119.394,E2 -3119.394} C_VEL
LIN {X 0,Y 552.112,Z 200.713,A -85,B 0,C 180,E1 -3121.905,E2 -3121.905} C_VEL
LIN {X 0,Y 552.145,Z 200.702,A -85,B 0,C 180,E1 -3124.652,E2 -3124.652} C_VEL
LIN {X 0,Y 552.086,Z 200.718,A -85,B 0,C 180,E1 -3127.551,E2 -3127.551} C_VEL
LIN {X 0,Y 552.141,Z 200.703,A -85,B 0,C 180,E1 -3130.376,E2 -3130.376} C_VEL
LIN {X 0,Y 552.149,Z 200.703,A -85,B 0,C 180,E1 -3132.979,E2 -3132.979} C_VEL
LIN {X 0,Y 552.131,Z 200.706,A -85,B 0,C 180,E1 -3136.006,E2 -3136.006} C_VEL
LIN {X 0,Y 552.16,Z 200.703,A -85,B 0,C 180,E1 -3138.995,E2 -3138.995} C_VEL
LIN {X 0,Y 552.155,Z 200.702,A -85,B 0,C 180,E1 -3141.952,E2 -3141.952} C_VEL
LIN {X 0,Y 552.228,Z 200.695,A -85,B 0,C 180,E1 -3144.89,E2 -3144.89} C_VEL
LIN {X 0,Y 552.227,Z 200.694,A -85,B 0,C 180,E1 -3147.812,E2 -3147.812} C_VEL
LIN {X 0,Y 552.238,Z 200.693,A -85,B 0,C 180,E1 -3150.729,E2 -3150.729} C_VEL
LIN {X 0,Y 552.201,Z 200.701,A -85,B 0,C 180,E1 -3152.918,E2 -3152.918} C_VEL
LIN {X 0,Y 552.199,Z 200.696,A -85,B 0,C 180,E1 -3155.843,E2 -3155.843} C_VEL
LIN {X 0,Y 552.156,Z 200.706,A -85,B 0,C 180,E1 -3158.785,E2 -3158.785} C_VEL
LIN {X 0,Y 552.16,Z 200.701,A -85,B 0,C 180,E1 -3161.749,E2 -3161.749} C_VEL
LIN {X 0,Y 552.132,Z 200.71,A -85,B 0,C 180,E1 -3164.747,E2 -3164.747} C_VEL
LIN {X 0,Y 552.108,Z 200.706,A -85,B 0,C 180,E1 -3167.787,E2 -3167.787} C_VEL
LIN {X 0,Y 552.125,Z 200.705,A -85,B 0,C 180,E1 -3170.099,E2 -3170.099} C_VEL
LIN {X 0,Y 552.088,Z 200.714,A -85,B 0,C 180,E1 -3172.449,E2 -3172.449} C_VEL
LIN {X 0,Y 552.146,Z 200.704,A -85,B 0,C 180,E1 -3175.349,E2 -3175.349} C_VEL
LIN {X 0,Y 552.115,Z 200.709,A -85,B 0,C 180,E1 -3178.095,E2 -3178.095} C_VEL
LIN {X 0,Y 552.157,Z 200.709,A -85,B 0,C 180,E1 -3181.027,E2 -3181.027} C_VEL
LIN {X 0,Y 552.194,Z 200.803,A -85,B 0,C 180,E1 -3181.451,E2 -3181.451} C_VEL
LIN {X 0,Y 552.368,Z 206.719,A -85,B 0,C 180,E1 -3182.587,E2 -3182.587} C_VEL
LIN {X 0,Y 552.178,Z 222.892,A -85,B 0,C 180,E1 -3185.681,E2 -3185.681} C_VEL
LIN {X 0,Y 553.399,Z 231.364,A -85,B 0,C 180,E1 -3185.839,E2 -3185.839} C_VEL
LIN {X 0,Y 553.085,Z 329.529,A -85,B 0,C 180,E1 -3187.139,E2 -3187.139} C_VEL
LIN {X 0,Y 552.913,Z 342.775,A -85,B 0,C 180,E1 -3187.463,E2 -3187.463} C_VEL
LIN {X 0,Y 552.834,Z 354.793,A -85,B 0,C 180,E1 -3187.903,E2 -3187.903} C_VEL
LIN {X 0,Y 552.664,Z 366.148,A -85,B 0,C 180,E1 -3188.461,E2 -3188.461} C_VEL
LIN {X 0,Y 552.451,Z 377.719,A -85,B 0,C 180,E1 -3189.19,E2 -3189.19} C_VEL
LIN {X 0,Y 552.279,Z 387.781,A -85,B 0,C 180,E1 -3189.983,E2 -3189.983} C_VEL
LIN {X 0,Y 552.128,Z 397.698,A -85,B 0,C 180,E1 -3190.955,E2 -3190.955} C_VEL
LIN {X 0,Y 551.978,Z 405.761,A -85,B 0,C 180,E1 -3191.917,E2 -3191.917} C_VEL
LIN {X 0,Y 551.851,Z 412.828,A -85,B 0,C 180,E1 -3192.943,E2 -3192.943} C_VEL
LIN {X 0,Y 551.833,Z 418.473,A -85,B 0,C 180,E1 -3193.949,E2 -3193.949} C_VEL
LIN {X 0,Y 551.767,Z 423.303,A -85,B 0,C 180,E1 -3195.016,E2 -3195.016} C_VEL
LIN {X 0,Y 551.72,Z 426.913,A -85,B 0,C 180,E1 -3196.034,E2 -3196.034} C_VEL
LIN {X 0,Y 551.672,Z 429.611,A -85,B 0,C 180,E1 -3197.043,E2 -3197.043} C_VEL
LIN {X 0,Y 551.663,Z 430.813,A -85,B 0,C 180,E1 -3197.631,E2 -3197.631} C_VEL
LIN {X 0,Y 551.651,Z 432.335,A -85,B 0,C 180,E1 -3198.727,E2 -3198.727} C_VEL
LIN {X 0,Y 551.647,Z 432.964,A -85,B 0,C 180,E1 -3199.846,E2 -3199.846} C_VEL
LIN {X 0,Y 551.638,Z 432.644,A -85,B 0,C 180,E1 -3200.993,E2 -3200.993} C_VEL
LIN {X 0,Y 551.674,Z 431.098,A -85,B 0,C 180,E1 -3202.303,E2 -3202.303} C_VEL
LIN {X 0,Y 551.744,Z 427.793,A -85,B 0,C 180,E1 -3203.753,E2 -3203.753} C_VEL
LIN {X 0,Y 551.713,Z 423.499,A -85,B 0,C 180,E1 -3205.024,E2 -3205.024} C_VEL
LIN {X 0,Y 551.815,Z 417.335,A -85,B 0,C 180,E1 -3206.357,E2 -3206.357} C_VEL
LIN {X 0,Y 551.884,Z 411.032,A -85,B 0,C 180,E1 -3207.426,E2 -3207.426} C_VEL
LIN {X 0,Y 552.033,Z 402.928,A -85,B 0,C 180,E1 -3208.535,E2 -3208.535} C_VEL
LIN {X 0,Y 552.169,Z 393.8,A -85,B 0,C 180,E1 -3209.541,E2 -3209.541} C_VEL
LIN {X 0,Y 552.356,Z 383.58,A -85,B 0,C 180,E1 -3210.46,E2 -3210.46} C_VEL
LIN {X 0,Y 552.531,Z 372.188,A -85,B 0,C 180,E1 -3211.272,E2 -3211.272} C_VEL
LIN {X 0,Y 552.777,Z 360.24,A -85,B 0,C 180,E1 -3211.939,E2 -3211.939} C_VEL
LIN {X 0,Y 552.932,Z 347.719,A -85,B 0,C 180,E1 -3212.462,E2 -3212.462} C_VEL
LIN {X 0,Y 553.021,Z 334.661,A -85,B 0,C 180,E1 -3212.845,E2 -3212.845} C_VEL
LIN {X 0,Y 553.129,Z 320.669,A -85,B 0,C 180,E1 -3213.087,E2 -3213.087} C_VEL
LIN {X 0,Y 553.403,Z 229.988,A -85,B 0,C 180,E1 -3214.268,E2 -3214.268} C_VEL
LIN {X 0,Y 552.192,Z 222.867,A -85,B 0,C 180,E1 -3214.407,E2 -3214.407} C_VEL
LIN {X 0,Y 552.246,Z 209.936,A -85,B 0,C 180,E1 -3216.765,E2 -3216.765} C_VEL
LIN {X 0,Y 552.12,Z 200.711,A -85,B 0,C 180,E1 -3218.388,E2 -3218.388} C_VEL
LIN {X 0,Y 552.089,Z 200.719,A -85,B 0,C 180,E1 -3221.443,E2 -3221.443} C_VEL
LIN {X 0,Y 552.086,Z 200.715,A -85,B 0,C 180,E1 -3223.737,E2 -3223.737} C_VEL
LIN {X 0,Y 552.092,Z 200.712,A -85,B 0,C 180,E1 -3226.004,E2 -3226.004} C_VEL
LIN {X 0,Y 552.158,Z 200.708,A -85,B 0,C 180,E1 -3228.994,E2 -3228.994} C_VEL
LIN {X 0,Y 552.112,Z 200.708,A -85,B 0,C 180,E1 -3231.951,E2 -3231.951} C_VEL
LIN {X 0,Y 552.153,Z 200.702,A -85,B 0,C 180,E1 -3234.156,E2 -3234.156} C_VEL
LIN {X 0,Y 552.162,Z 200.709,A -85,B 0,C 180,E1 -3237.082,E2 -3237.082} C_VEL
LIN {X 0,Y 552.168,Z 200.7,A -85,B 0,C 180,E1 -3240,E2 -3240} C_VEL
LIN {X 0,Y 552.159,Z 200.709,A -85,B 0,C 180,E1 -3242.919,E2 -3242.919} C_VEL
LIN {X 0,Y 552.143,Z 200.702,A -85,B 0,C 180,E1 -3245.845,E2 -3245.845} C_VEL
LIN {X 0,Y 552.115,Z 200.714,A -85,B 0,C 180,E1 -3248.787,E2 -3248.787} C_VEL
LIN {X 0,Y 552.112,Z 200.706,A -85,B 0,C 180,E1 -3251.752,E2 -3251.752} C_VEL
LIN {X 0,Y 552.083,Z 200.718,A -85,B 0,C 180,E1 -3254.75,E2 -3254.75} C_VEL
LIN {X 0,Y 552.091,Z 200.708,A -85,B 0,C 180,E1 -3257.789,E2 -3257.789} C_VEL
LIN {X 0,Y 552.086,Z 200.711,A -85,B 0,C 180,E1 -3260.103,E2 -3260.103} C_VEL
LIN {X 0,Y 552.065,Z 200.719,A -85,B 0,C 180,E1 -3262.452,E2 -3262.452} C_VEL
LIN {X 0,Y 552.109,Z 200.707,A -85,B 0,C 180,E1 -3265.353,E2 -3265.353} C_VEL
LIN {X 0,Y 552.089,Z 200.712,A -85,B 0,C 180,E1 -3268.1,E2 -3268.1} C_VEL
LIN {X 0,Y 552.065,Z 200.72,A -85,B 0,C 180,E1 -3270.612,E2 -3270.612} C_VEL
LIN {X 0,Y 552.081,Z 200.711,A -85,B 0,C 180,E1 -3273.188,E2 -3273.188} C_VEL
LIN {X 0,Y 552.075,Z 200.712,A -85,B 0,C 180,E1 -3275.845,E2 -3275.845} C_VEL
LIN {X 0,Y 552.088,Z 200.71,A -85,B 0,C 180,E1 -3279.065,E2 -3279.065} C_VEL
LIN {X 0,Y 552.107,Z 200.707,A -85,B 0,C 180,E1 -3281.448,E2 -3281.448} C_VEL
LIN {X 0,Y 552.066,Z 200.716,A -85,B 0,C 180,E1 -3284.535,E2 -3284.535} C_VEL
LIN {X 0,Y 552.106,Z 200.709,A -85,B 0,C 180,E1 -3287.588,E2 -3287.588} C_VEL
LIN {X 0,Y 552.109,Z 200.711,A -85,B 0,C 180,E1 -3290.476,E2 -3290.476} C_VEL
LIN {X 0,Y 552.095,Z 200.71,A -85,B 0,C 180,E1 -3293.319,E2 -3293.319} C_VEL
LIN {X 0,Y 552.112,Z 200.715,A -85,B 0,C 180,E1 -3295.942,E2 -3295.942} C_VEL
LIN {X 0,Y 552.106,Z 200.71,A -85,B 0,C 180,E1 -3298.544,E2 -3298.544} C_VEL
LIN {X 0,Y 552.113,Z 200.711,A -85,B 0,C 180,E1 -3301.441,E2 -3301.441} C_VEL
LIN {X 0,Y 552.121,Z 200.71,A -85,B 0,C 180,E1 -3304.358,E2 -3304.358} C_VEL
LIN {X 0,Y 552.142,Z 200.737,A -85,B 0,C 180,E1 -3305.817,E2 -3305.817} C_VEL
LIN {X 0,Y 553.1,Z 207.419,A -85,B 0,C 180,E1 -3306.805,E2 -3306.805} C_VEL
LIN {X 0,Y 552.868,Z 228.013,A -85,B 0,C 180,E1 -3309.735,E2 -3309.735} C_VEL
LIN {X 0,Y 552.599,Z 249.583,A -85,B 0,C 180,E1 -3312.761,E2 -3312.761} C_VEL
LIN {X 0,Y 552.374,Z 270.218,A -85,B 0,C 180,E1 -3315.626,E2 -3315.626} C_VEL
LIN {X 0,Y 553.366,Z 278.442,A -85,B 0,C 180,E1 -3315.762,E2 -3315.762} C_VEL
LIN {X 0,Y 553.1,Z 378.867,A -85,B 0,C 180,E1 -3317.083,E2 -3317.083} C_VEL
LIN {X 0,Y 552.967,Z 392.184,A -85,B 0,C 180,E1 -3317.407,E2 -3317.407} C_VEL
LIN {X 0,Y 552.805,Z 405.18,A -85,B 0,C 180,E1 -3317.878,E2 -3317.878} C_VEL
LIN {X 0,Y 552.682,Z 417.646,A -85,B 0,C 180,E1 -3318.507,E2 -3318.507} C_VEL
LIN {X 0,Y 552.469,Z 429.5,A -85,B 0,C 180,E1 -3319.279,E2 -3319.279} C_VEL
LIN {X 0,Y 552.283,Z 439.657,A -85,B 0,C 180,E1 -3320.109,E2 -3320.109} C_VEL
LIN {X 0,Y 552.103,Z 448.794,A -85,B 0,C 180,E1 -3321.03,E2 -3321.03} C_VEL
LIN {X 0,Y 551.959,Z 457.694,A -85,B 0,C 180,E1 -3322.134,E2 -3322.134} C_VEL
LIN {X 0,Y 551.835,Z 464.852,A -85,B 0,C 180,E1 -3323.235,E2 -3323.235} C_VEL
LIN {X 0,Y 551.804,Z 471.368,A -85,B 0,C 180,E1 -3324.519,E2 -3324.519} C_VEL
LIN {X 0,Y 551.764,Z 475.678,A -85,B 0,C 180,E1 -3325.617,E2 -3325.617} C_VEL
LIN {X 0,Y 551.75,Z 477.959,A -85,B 0,C 180,E1 -3326.349,E2 -3326.349} C_VEL
LIN {X 0,Y 551.723,Z 479.807,A -85,B 0,C 180,E1 -3327.08,E2 -3327.08} C_VEL
LIN {X 0,Y 551.645,Z 482.183,A -85,B 0,C 180,E1 -3328.54,E2 -3328.54} C_VEL
LIN {X 0,Y 551.64,Z 483,A -85,B 0,C 180,E1 -3330,E2 -3330} C_VEL
LIN {X 0,Y 551.645,Z 482.184,A -85,B 0,C 180,E1 -3331.46,E2 -3331.46} C_VEL
LIN {X 0,Y 551.723,Z 479.811,A -85,B 0,C 180,E1 -3332.92,E2 -3332.92} C_VEL
LIN {X 0,Y 551.764,Z 476.897,A -85,B 0,C 180,E1 -3334.017,E2 -3334.017} C_VEL
LIN {X 0,Y 551.723,Z 472.951,A -85,B 0,C 180,E1 -3335.115,E2 -3335.115} C_VEL
LIN {X 0,Y 551.814,Z 467.129,A -85,B 0,C 180,E1 -3336.352,E2 -3336.352} C_VEL
LIN {X 0,Y 551.926,Z 460.241,A -85,B 0,C 180,E1 -3337.499,E2 -3337.499} C_VEL
LIN {X 0,Y 552.081,Z 452,A -85,B 0,C 180,E1 -3338.601,E2 -3338.601} C_VEL
LIN {X 0,Y 552.224,Z 443.551,A -85,B 0,C 180,E1 -3339.522,E2 -3339.522} C_VEL
LIN {X 0,Y 552.427,Z 433.106,A -85,B 0,C 180,E1 -3340.444,E2 -3340.444} C_VEL
LIN {X 0,Y 552.592,Z 422.146,A -85,B 0,C 180,E1 -3341.223,E2 -3341.223} C_VEL
LIN {X 0,Y 552.749,Z 411.43,A -85,B 0,C 180,E1 -3341.829,E2 -3341.829} C_VEL
LIN {X 0,Y 552.887,Z 399.769,A -85,B 0,C 180,E1 -3342.338,E2 -3342.338} C_VEL
LIN {X 0,Y 553.06,Z 387.225,A -85,B 0,C 180,E1 -3342.731,E2 -3342.731} C_VEL
LIN {X 0,Y 553.139,Z 374.536,A -85,B 0,C 180,E1 -3342.986,E2 -3342.986} C_VEL
LIN {X 0,Y 553.258,Z 276.372,A -85,B 0,C 180,E1 -3344.268,E2 -3344.268} C_VEL
LIN {X 0,Y 552.397,Z 270.262,A -85,B 0,C 180,E1 -3344.385,E2 -3344.385} C_VEL
LIN {X 0,Y 552.619,Z 249.901,A -85,B 0,C 180,E1 -3347.24,E2 -3347.24} C_VEL
LIN {X 0,Y 552.943,Z 228.599,A -85,B 0,C 180,E1 -3350.262,E2 -3350.262} C_VEL
LIN {X 0,Y 553.296,Z 208.329,A -85,B 0,C 180,E1 -3353.186,E2 -3353.186} C_VEL
LIN {X 0,Y 552.136,Z 200.712,A -85,B 0,C 180,E1 -3354.383,E2 -3354.383} C_VEL
LIN {X 0,Y 552.115,Z 200.708,A -85,B 0,C 180,E1 -3357.271,E2 -3357.271} C_VEL
LIN {X 0,Y 552.106,Z 200.716,A -85,B 0,C 180,E1 -3360.048,E2 -3360.048} C_VEL
LIN {X 0,Y 552.101,Z 200.708,A -85,B 0,C 180,E1 -3362.843,E2 -3362.843} C_VEL
LIN {X 0,Y 552.08,Z 200.712,A -85,B 0,C 180,E1 -3365.44,E2 -3365.44} C_VEL
LIN {X 0,Y 552.077,Z 200.72,A -85,B 0,C 180,E1 -3367.883,E2 -3367.883} C_VEL
LIN {X 0,Y 552.097,Z 200.71,A -85,B 0,C 180,E1 -3370.477,E2 -3370.477} C_VEL
LIN {X 0,Y 552.077,Z 200.715,A -85,B 0,C 180,E1 -3373.48,E2 -3373.48} C_VEL
LIN {X 0,Y 552.09,Z 200.709,A -85,B 0,C 180,E1 -3376.574,E2 -3376.574} C_VEL
LIN {X 0,Y 552.087,Z 200.716,A -85,B 0,C 180,E1 -3379.517,E2 -3379.517} C_VEL
LIN {X 0,Y 552.056,Z 200.714,A -85,B 0,C 180,E1 -3382.333,E2 -3382.333} C_VEL
LIN {X 0,Y 552.092,Z 200.711,A -85,B 0,C 180,E1 -3385.051,E2 -3385.051} C_VEL
LIN {X 0,Y 552.088,Z 200.717,A -85,B 0,C 180,E1 -3387.679,E2 -3387.679} C_VEL
LIN {X 0,Y 552.069,Z 200.712,A -85,B 0,C 180,E1 -3390.232,E2 -3390.232} C_VEL
LIN {X 0,Y 552.1,Z 200.71,A -85,B 0,C 180,E1 -3392.995,E2 -3392.995} C_VEL
LIN {X 0,Y 552.066,Z 200.717,A -85,B 0,C 180,E1 -3395.159,E2 -3395.159} C_VEL
LIN {X 0,Y 552.065,Z 200.719,A -85,B 0,C 180,E1 -3397.548,E2 -3397.548} C_VEL
LIN {X 0,Y 552.106,Z 200.708,A -85,B 0,C 180,E1 -3400.672,E2 -3400.672} C_VEL
LIN {X 0,Y 552.14,Z 200.708,A -85,B 0,C 180,E1 -3402.977,E2 -3402.977} C_VEL
LIN {X 0,Y 552.082,Z 200.71,A -85,B 0,C 180,E1 -3406.003,E2 -3406.003} C_VEL
LIN {X 0,Y 552.155,Z 200.708,A -85,B 0,C 180,E1 -3408.993,E2 -3408.993} C_VEL
LIN {X 0,Y 552.108,Z 200.707,A -85,B 0,C 180,E1 -3411.951,E2 -3411.951} C_VEL
LIN {X 0,Y 552.179,Z 200.705,A -85,B 0,C 180,E1 -3414.888,E2 -3414.888} C_VEL
LIN {X 0,Y 552.161,Z 200.7,A -85,B 0,C 180,E1 -3417.811,E2 -3417.811} C_VEL
LIN {X 0,Y 552.197,Z 200.702,A -85,B 0,C 180,E1 -3420.729,E2 -3420.729} C_VEL
LIN {X 0,Y 552.161,Z 200.709,A -85,B 0,C 180,E1 -3422.918,E2 -3422.918} C_VEL
LIN {X 0,Y 552.153,Z 200.701,A -85,B 0,C 180,E1 -3425.844,E2 -3425.844} C_VEL
LIN {X 0,Y 552.111,Z 200.707,A -85,B 0,C 180,E1 -3428.049,E2 -3428.049} C_VEL
LIN {X 0,Y 552.157,Z 200.706,A -85,B 0,C 180,E1 -3431.006,E2 -3431.006} C_VEL
LIN {X 0,Y 552.091,Z 200.71,A -85,B 0,C 180,E1 -3433.996,E2 -3433.996} C_VEL
LIN {X 0,Y 552.143,Z 200.703,A -85,B 0,C 180,E1 -3437.343,E2 -3437.343} C_VEL
LIN {X 0,Y 552.089,Z 200.712,A -85,B 0,C 180,E1 -3440.103,E2 -3440.103} C_VEL
LIN {X 0,Y 552.11,Z 200.715,A -85,B 0,C 180,E1 -3442.45,E2 -3442.45} C_VEL
LIN {X 0,Y 552.112,Z 200.706,A -85,B 0,C 180,E1 -3445.354,E2 -3445.354} C_VEL
LIN {X 0,Y 552.094,Z 200.713,A -85,B 0,C 180,E1 -3448.099,E2 -3448.099} C_VEL
LIN {X 0,Y 552.068,Z 200.716,A -85,B 0,C 180,E1 -3450.659,E2 -3450.659} C_VEL
LIN {X 0,Y 552.087,Z 200.709,A -85,B 0,C 180,E1 -3453.187,E2 -3453.187} C_VEL
LIN {X 0,Y 552.084,Z 200.713,A -85,B 0,C 180,E1 -3453.84,E2 -3453.84} C_VEL
LIN {X 0,Y 551.452,Z 200.798,A -85,B 0,C 180,E1 -3454.448,E2 -3454.448} C_VEL
LIN {X 0,Y 548.625,Z 201.149,A -85,B 0,C 180,E1 -3455.436,E2 -3455.436} C_VEL
LIN {X 0,Y 546.198,Z 201.453,A -85,B 0,C 180,E1 -3456.232,E2 -3456.232} C_VEL
LIN {X 0,Y 545.127,Z 201.578,A -85,B 0,C 180,E1 -3456.846,E2 -3456.846} C_VEL
LIN {X 0,Y 545.025,Z 201.589,A -85,B 0,C 180,E1 -3457.054,E2 -3457.054} C_VEL
LIN {X 0,Y 545.068,Z 201.593,A -85,B 0,C 180,E1 -3460.142,E2 -3460.142} C_VEL
LIN {X 0,Y 545.034,Z 201.589,A -85,B 0,C 180,E1 -3462.7,E2 -3462.7} C_VEL
LIN {X 0,Y 545.031,Z 201.588,A -85,B 0,C 180,E1 -3465.17,E2 -3465.17} C_VEL
LIN {X 0,Y 545.056,Z 201.593,A -85,B 0,C 180,E1 -3467.901,E2 -3467.901} C_VEL
LIN {X 0,Y 545.081,Z 201.583,A -85,B 0,C 180,E1 -3470.679,E2 -3470.679} C_VEL
LIN {X 0,Y 545.033,Z 201.593,A -85,B 0,C 180,E1 -3473.624,E2 -3473.624} C_VEL
LIN {X 0,Y 545.058,Z 201.587,A -85,B 0,C 180,E1 -3476.332,E2 -3476.332} C_VEL
LIN {X 0,Y 545.053,Z 201.586,A -85,B 0,C 180,E1 -3478.955,E2 -3478.955} C_VEL
LIN {X 0,Y 545.089,Z 201.587,A -85,B 0,C 180,E1 -3481.511,E2 -3481.511} C_VEL
LIN {X 0,Y 545.088,Z 201.581,A -85,B 0,C 180,E1 -3484.492,E2 -3484.492} C_VEL
LIN {X 0,Y 545.034,Z 201.591,A -85,B 0,C 180,E1 -3487.245,E2 -3487.245} C_VEL
LIN {X 0,Y 545.113,Z 201.578,A -85,B 0,C 180,E1 -3490.417,E2 -3490.417} C_VEL
LIN {X 0,Y 545.068,Z 201.593,A -85,B 0,C 180,E1 -3493.523,E2 -3493.523} C_VEL
LIN {X 0,Y 545.09,Z 201.585,A -85,B 0,C 180,E1 -3495.821,E2 -3495.821} C_VEL
LIN {X 0,Y 545.115,Z 201.579,A -85,B 0,C 180,E1 -3498.851,E2 -3498.851} C_VEL
LIN {X 0,Y 545.126,Z 201.579,A -85,B 0,C 180,E1 -3501.848,E2 -3501.848} C_VEL
LIN {X 0,Y 545.203,Z 201.569,A -85,B 0,C 180,E1 -3504.824,E2 -3504.824} C_VEL
LIN {X 0,Y 545.198,Z 201.569,A -85,B 0,C 180,E1 -3507.784,E2 -3507.784} C_VEL
LIN {X 0,Y 545.209,Z 201.569,A -85,B 0,C 180,E1 -3510.739,E2 -3510.739} C_VEL
LIN {X 0,Y 545.169,Z 201.577,A -85,B 0,C 180,E1 -3512.956,E2 -3512.956} C_VEL
LIN {X 0,Y 545.169,Z 201.571,A -85,B 0,C 180,E1 -3515.919,E2 -3515.919} C_VEL
LIN {X 0,Y 545.115,Z 201.585,A -85,B 0,C 180,E1 -3518.899,E2 -3518.899} C_VEL
LIN {X 0,Y 545.132,Z 201.576,A -85,B 0,C 180,E1 -3521.903,E2 -3521.903} C_VEL
LIN {X 0,Y 545.081,Z 201.591,A -85,B 0,C 180,E1 -3524.942,E2 -3524.942} C_VEL
LIN {X 0,Y 545.076,Z 201.583,A -85,B 0,C 180,E1 -3528.024,E2 -3528.024} C_VEL
LIN {X 0,Y 545.091,Z 201.584,A -85,B 0,C 180,E1 -3530.37,E2 -3530.37} C_VEL
LIN {X 0,Y 545.082,Z 201.582,A -85,B 0,C 180,E1 -3533.557,E2 -3533.557} C_VEL
LIN {X 0,Y 545.079,Z 201.584,A -85,B 0,C 180,E1 -3535.998,E2 -3535.998} C_VEL
LIN {X 0,Y 545.08,Z 201.591,A -85,B 0,C 180,E1 -3538.747,E2 -3538.747} C_VEL
LIN {X 0,Y 545.145,Z 201.588,A -85,B 0,C 180,E1 -3541.349,E2 -3541.349} C_VEL
LIN {X 0,Y 545.358,Z 207.736,A -85,B 0,C 180,E1 -3542.546,E2 -3542.546} C_VEL
LIN {X 0,Y 545.172,Z 223.134,A -85,B 0,C 180,E1 -3545.496,E2 -3545.496} C_VEL
LIN {X 0,Y 546.518,Z 231.384,A -85,B 0,C 180,E1 -3545.655,E2 -3545.655} C_VEL
LIN {X 0,Y 546.188,Z 329.731,A -85,B 0,C 180,E1 -3546.976,E2 -3546.976} C_VEL
LIN {X 0,Y 545.991,Z 343.179,A -85,B 0,C 180,E1 -3547.31,E2 -3547.31} C_VEL
LIN {X 0,Y 545.895,Z 355.136,A -85,B 0,C 180,E1 -3547.753,E2 -3547.753} C_VEL
LIN {X 0,Y 545.701,Z 367.015,A -85,B 0,C 180,E1 -3548.349,E2 -3548.349} C_VEL
LIN {X 0,Y 545.5,Z 377.555,A -85,B 0,C 180,E1 -3549.022,E2 -3549.022} C_VEL
LIN {X 0,Y 545.288,Z 387.561,A -85,B 0,C 180,E1 -3549.812,E2 -3549.812} C_VEL
LIN {X 0,Y 545.088,Z 397.349,A -85,B 0,C 180,E1 -3550.77,E2 -3550.77} C_VEL
LIN {X 0,Y 544.949,Z 406.049,A -85,B 0,C 180,E1 -3551.821,E2 -3551.821} C_VEL
LIN {X 0,Y 544.794,Z 413.133,A -85,B 0,C 180,E1 -3552.871,E2 -3552.871} C_VEL
LIN {X 0,Y 544.749,Z 418.881,A -85,B 0,C 180,E1 -3553.924,E2 -3553.924} C_VEL
LIN {X 0,Y 544.668,Z 424.345,A -85,B 0,C 180,E1 -3555.202,E2 -3555.202} C_VEL
LIN {X 0,Y 544.612,Z 427.808,A -85,B 0,C 180,E1 -3556.268,E2 -3556.268} C_VEL
LIN {X 0,Y 544.591,Z 430.385,A -85,B 0,C 180,E1 -3557.35,E2 -3557.35} C_VEL
LIN {X 0,Y 544.548,Z 432.497,A -85,B 0,C 180,E1 -3558.837,E2 -3558.837} C_VEL
LIN {X 0,Y 544.547,Z 432.98,A -85,B 0,C 180,E1 -3559.812,E2 -3559.812} C_VEL
LIN {X 0,Y 544.536,Z 432.817,A -85,B 0,C 180,E1 -3560.772,E2 -3560.772} C_VEL
LIN {X 0,Y 544.541,Z 431.739,A -85,B 0,C 180,E1 -3561.924,E2 -3561.924} C_VEL
LIN {X 0,Y 544.579,Z 429.55,A -85,B 0,C 180,E1 -3563.134,E2 -3563.134} C_VEL
LIN {X 0,Y 544.635,Z 425.729,A -85,B 0,C 180,E1 -3564.502,E2 -3564.502} C_VEL
LIN {X 0,Y 544.645,Z 421.232,A -85,B 0,C 180,E1 -3565.665,E2 -3565.665} C_VEL
LIN {X 0,Y 544.792,Z 414.564,A -85,B 0,C 180,E1 -3566.975,E2 -3566.975} C_VEL
LIN {X 0,Y 544.899,Z 407.496,A -85,B 0,C 180,E1 -3568.075,E2 -3568.075} C_VEL
LIN {X 0,Y 545.109,Z 398.597,A -85,B 0,C 180,E1 -3569.184,E2 -3569.184} C_VEL
LIN {X 0,Y 545.286,Z 389.072,A -85,B 0,C 180,E1 -3570.144,E2 -3570.144} C_VEL
LIN {X 0,Y 545.428,Z 379.115,A -85,B 0,C 180,E1 -3570.96,E2 -3570.96} C_VEL
LIN {X 0,Y 545.652,Z 368.748,A -85,B 0,C 180,E1 -3571.644,E2 -3571.644} C_VEL
LIN {X 0,Y 545.911,Z 356.293,A -85,B 0,C 180,E1 -3572.286,E2 -3572.286} C_VEL
LIN {X 0,Y 546.047,Z 343.637,A -85,B 0,C 180,E1 -3572.766,E2 -3572.766} C_VEL
LIN {X 0,Y 546.194,Z 330.385,A -85,B 0,C 180,E1 -3573.101,E2 -3573.101} C_VEL
LIN {X 0,Y 546.479,Z 253.667,A -85,B 0,C 180,E1 -3574.138,E2 -3574.138} C_VEL
LIN {X 0,Y 546.393,Z 229.692,A -85,B 0,C 180,E1 -3574.459,E2 -3574.459} C_VEL
LIN {X 0,Y 545.158,Z 223.062,A -85,B 0,C 180,E1 -3574.597,E2 -3574.597} C_VEL
LIN {X 0,Y 545.21,Z 209.454,A -85,B 0,C 180,E1 -3577.05,E2 -3577.05} C_VEL
LIN {X 0,Y 545.099,Z 201.585,A -85,B 0,C 180,E1 -3578.438,E2 -3578.438} C_VEL
LIN {X 0,Y 545.04,Z 201.595,A -85,B 0,C 180,E1 -3581.194,E2 -3581.194} C_VEL
LIN {X 0,Y 545.047,Z 201.595,A -85,B 0,C 180,E1 -3583.521,E2 -3583.521} C_VEL
LIN {X 0,Y 545.04,Z 201.59,A -85,B 0,C 180,E1 -3586.58,E2 -3586.58} C_VEL
LIN {X 0,Y 545.104,Z 201.585,A -85,B 0,C 180,E1 -3588.849,E2 -3588.849} C_VEL
LIN {X 0,Y 545.082,Z 201.585,A -85,B 0,C 180,E1 -3591.847,E2 -3591.847} C_VEL
LIN {X 0,Y 545.125,Z 201.577,A -85,B 0,C 180,E1 -3594.08,E2 -3594.08} C_VEL
LIN {X 0,Y 545.128,Z 201.585,A -85,B 0,C 180,E1 -3597.044,E2 -3597.044} C_VEL
LIN {X 0,Y 545.139,Z 201.576,A -85,B 0,C 180,E1 -3600,E2 -3600} C_VEL
LIN {X 0,Y 545.125,Z 201.586,A -85,B 0,C 180,E1 -3602.956,E2 -3602.956} C_VEL
LIN {X 0,Y 545.114,Z 201.577,A -85,B 0,C 180,E1 -3605.92,E2 -3605.92} C_VEL
LIN {X 0,Y 545.073,Z 201.591,A -85,B 0,C 180,E1 -3608.901,E2 -3608.901} C_VEL
LIN {X 0,Y 545.082,Z 201.582,A -85,B 0,C 180,E1 -3611.906,E2 -3611.906} C_VEL
LIN {X 0,Y 545.033,Z 201.595,A -85,B 0,C 180,E1 -3614.945,E2 -3614.945} C_VEL
LIN {X 0,Y 545.091,Z 201.581,A -85,B 0,C 180,E1 -3617.447,E2 -3617.447} C_VEL
LIN {X 0,Y 545.051,Z 201.591,A -85,B 0,C 180,E1 -3620.374,E2 -3620.374} C_VEL
LIN {X 0,Y 545.066,Z 201.583,A -85,B 0,C 180,E1 -3623.56,E2 -3623.56} C_VEL
LIN {X 0,Y 545.042,Z 201.589,A -85,B 0,C 180,E1 -3626.003,E2 -3626.003} C_VEL
LIN {X 0,Y 545.053,Z 201.591,A -85,B 0,C 180,E1 -3628.752,E2 -3628.752} C_VEL
LIN {X 0,Y 545.032,Z 201.59,A -85,B 0,C 180,E1 -3631.917,E2 -3631.917} C_VEL
LIN {X 0,Y 545.042,Z 201.593,A -85,B 0,C 180,E1 -3634.566,E2 -3634.566} C_VEL
LIN {X 0,Y 545.005,Z 201.592,A -85,B 0,C 180,E1 -3637.307,E2 -3637.307} C_VEL
LIN {X 0,Y 545.039,Z 201.595,A -85,B 0,C 180,E1 -3640.145,E2 -3640.145} C_VEL
LIN {X 0,Y 545.033,Z 201.59,A -85,B 0,C 180,E1 -3642.7,E2 -3642.7} C_VEL
LIN {X 0,Y 545.009,Z 201.591,A -85,B 0,C 180,E1 -3645.173,E2 -3645.173} C_VEL
LIN {X 0,Y 545.059,Z 201.591,A -85,B 0,C 180,E1 -3647.901,E2 -3647.901} C_VEL
LIN {X 0,Y 545.06,Z 201.586,A -85,B 0,C 180,E1 -3650.822,E2 -3650.822} C_VEL
LIN {X 0,Y 545.035,Z 201.592,A -85,B 0,C 180,E1 -3653.624,E2 -3653.624} C_VEL
LIN {X 0,Y 545.051,Z 201.591,A -85,B 0,C 180,E1 -3656.331,E2 -3656.331} C_VEL
LIN {X 0,Y 545.054,Z 201.587,A -85,B 0,C 180,E1 -3658.955,E2 -3658.955} C_VEL
LIN {X 0,Y 545.09,Z 201.587,A -85,B 0,C 180,E1 -3661.51,E2 -3661.51} C_VEL
LIN {X 0,Y 545.087,Z 201.585,A -85,B 0,C 180,E1 -3664.494,E2 -3664.494} C_VEL
LIN {X 0,Y 545.121,Z 201.681,A -85,B 0,C 180,E1 -3665.698,E2 -3665.698} C_VEL
LIN {X 0,Y 546.139,Z 208.311,A -85,B 0,C 180,E1 -3666.693,E2 -3666.693} C_VEL
LIN {X 0,Y 545.872,Z 227.572,A -85,B 0,C 180,E1 -3669.464,E2 -3669.464} C_VEL
LIN {X 0,Y 545.573,Z 249.092,A -85,B 0,C 180,E1 -3672.524,E2 -3672.524} C_VEL
LIN {X 0,Y 545.31,Z 269.836,A -85,B 0,C 180,E1 -3675.434,E2 -3675.434} C_VEL
LIN {X 0,Y 546.472,Z 279.252,A -85,B 0,C 180,E1 -3675.598,E2 -3675.598} C_VEL
LIN {X 0,Y 546.176,Z 378.194,A -85,B 0,C 180,E1 -3676.917,E2 -3676.917} C_VEL
LIN {X 0,Y 546.019,Z 391.621,A -85,B 0,C 180,E1 -3677.244,E2 -3677.244} C_VEL
LIN {X 0,Y 545.823,Z 405.008,A -85,B 0,C 180,E1 -3677.735,E2 -3677.735} C_VEL
LIN {X 0,Y 545.692,Z 416.814,A -85,B 0,C 180,E1 -3678.332,E2 -3678.332} C_VEL
LIN {X 0,Y 545.475,Z 427.904,A -85,B 0,C 180,E1 -3679.046,E2 -3679.046} C_VEL
LIN {X 0,Y 545.264,Z 438.402,A -85,B 0,C 180,E1 -3679.887,E2 -3679.887} C_VEL
LIN {X 0,Y 545.084,Z 446.984,A -85,B 0,C 180,E1 -3680.726,E2 -3680.726} C_VEL
LIN {X 0,Y 544.977,Z 454.904,A -85,B 0,C 180,E1 -3681.659,E2 -3681.659} C_VEL
LIN {X 0,Y 544.823,Z 462.621,A -85,B 0,C 180,E1 -3682.775,E2 -3682.775} C_VEL
LIN {X 0,Y 544.776,Z 469.682,A -85,B 0,C 180,E1 -3684.077,E2 -3684.077} C_VEL
LIN {X 0,Y 544.628,Z 474.375,A -85,B 0,C 180,E1 -3685.189,E2 -3685.189} C_VEL
LIN {X 0,Y 544.669,Z 477.959,A -85,B 0,C 180,E1 -3686.301,E2 -3686.301} C_VEL
LIN {X 0,Y 544.65,Z 479.807,A -85,B 0,C 180,E1 -3687.042,E2 -3687.042} C_VEL
LIN {X 0,Y 544.546,Z 482.182,A -85,B 0,C 180,E1 -3688.521,E2 -3688.521} C_VEL
LIN {X 0,Y 544.541,Z 483,A -85,B 0,C 180,E1 -3690,E2 -3690} C_VEL
LIN {X 0,Y 544.546,Z 482.183,A -85,B 0,C 180,E1 -3691.479,E2 -3691.479} C_VEL
LIN {X 0,Y 544.65,Z 479.811,A -85,B 0,C 180,E1 -3692.958,E2 -3692.958} C_VEL
LIN {X 0,Y 544.684,Z 476.897,A -85,B 0,C 180,E1 -3694.069,E2 -3694.069} C_VEL
LIN {X 0,Y 544.653,Z 472.95,A -85,B 0,C 180,E1 -3695.182,E2 -3695.182} C_VEL
LIN {X 0,Y 544.729,Z 467.649,A -85,B 0,C 180,E1 -3696.339,E2 -3696.339} C_VEL
LIN {X 0,Y 544.836,Z 461.462,A -85,B 0,C 180,E1 -3697.411,E2 -3697.411} C_VEL
LIN {X 0,Y 545.006,Z 453.412,A -85,B 0,C 180,E1 -3698.527,E2 -3698.527} C_VEL
LIN {X 0,Y 545.125,Z 445.202,A -85,B 0,C 180,E1 -3699.46,E2 -3699.46} C_VEL
LIN {X 0,Y 545.374,Z 435.195,A -85,B 0,C 180,E1 -3700.393,E2 -3700.393} C_VEL
LIN {X 0,Y 545.542,Z 424.252,A -85,B 0,C 180,E1 -3701.211,E2 -3701.211} C_VEL
LIN {X 0,Y 545.739,Z 412.809,A -85,B 0,C 180,E1 -3701.889,E2 -3701.889} C_VEL
LIN {X 0,Y 545.901,Z 400.529,A -85,B 0,C 180,E1 -3702.452,E2 -3702.452} C_VEL
LIN {X 0,Y 546.11,Z 387.614,A -85,B 0,C 180,E1 -3702.872,E2 -3702.872} C_VEL
LIN {X 0,Y 546.203,Z 375.385,A -85,B 0,C 180,E1 -3703.13,E2 -3703.13} C_VEL
LIN {X 0,Y 546.444,Z 277.484,A -85,B 0,C 180,E1 -3704.427,E2 -3704.427} C_VEL
LIN {X 0,Y 545.362,Z 270.014,A -85,B 0,C 180,E1 -3704.569,E2 -3704.569} C_VEL
LIN {X 0,Y 545.606,Z 248.734,A -85,B 0,C 180,E1 -3707.597,E2 -3707.597} C_VEL
LIN {X 0,Y 545.962,Z 229.678,A -85,B 0,C 180,E1 -3710.336,E2 -3710.336} C_VEL
LIN {X 0,Y 546.351,Z 209.434,A -85,B 0,C 180,E1 -3713.298,E2 -3713.298} C_VEL
LIN {X 0,Y 545.092,Z 201.589,A -85,B 0,C 180,E1 -3714.542,E2 -3714.542} C_VEL
LIN {X 0,Y 545.067,Z 201.589,A -85,B 0,C 180,E1 -3717.654,E2 -3717.654} C_VEL
LIN {X 0,Y 545.065,Z 201.592,A -85,B 0,C 180,E1 -3720.243,E2 -3720.243} C_VEL
LIN {X 0,Y 545.065,Z 201.584,A -85,B 0,C 180,E1 -3723.059,E2 -3723.059} C_VEL
LIN {X 0,Y 545.037,Z 201.592,A -85,B 0,C 180,E1 -3725.673,E2 -3725.673} C_VEL
LIN {X 0,Y 545.032,Z 201.593,A -85,B 0,C 180,E1 -3728.234,E2 -3728.234} C_VEL
LIN {X 0,Y 545.073,Z 201.583,A -85,B 0,C 180,E1 -3731.11,E2 -3731.11} C_VEL
LIN {X 0,Y 545.028,Z 201.593,A -85,B 0,C 180,E1 -3734.126,E2 -3734.126} C_VEL
LIN {X 0,Y 545.057,Z 201.585,A -85,B 0,C 180,E1 -3736.891,E2 -3736.891} C_VEL
LIN {X 0,Y 545.056,Z 201.592,A -85,B 0,C 180,E1 -3739.856,E2 -3739.856} C_VEL
LIN {X 0,Y 545.042,Z 201.589,A -85,B 0,C 180,E1 -3743.069,E2 -3743.069} C_VEL
LIN {X 0,Y 545.051,Z 201.595,A -85,B 0,C 180,E1 -3745.602,E2 -3745.602} C_VEL
LIN {X 0,Y 545.036,Z 201.588,A -85,B 0,C 180,E1 -3748.314,E2 -3748.314} C_VEL
LIN {X 0,Y 545.067,Z 201.593,A -85,B 0,C 180,E1 -3751.505,E2 -3751.505} C_VEL
LIN {X 0,Y 545.051,Z 201.586,A -85,B 0,C 180,E1 -3754.488,E2 -3754.488} C_VEL
LIN {X 0,Y 545.018,Z 201.597,A -85,B 0,C 180,E1 -3757.241,E2 -3757.241} C_VEL
LIN {X 0,Y 545.069,Z 201.583,A -85,B 0,C 180,E1 -3760.413,E2 -3760.413} C_VEL
LIN {X 0,Y 545.096,Z 201.582,A -85,B 0,C 180,E1 -3762.75,E2 -3762.75} C_VEL
LIN {X 0,Y 545.04,Z 201.588,A -85,B 0,C 180,E1 -3765.818,E2 -3765.818} C_VEL
LIN {X 0,Y 545.102,Z 201.584,A -85,B 0,C 180,E1 -3768.849,E2 -3768.849} C_VEL
LIN {X 0,Y 545.078,Z 201.583,A -85,B 0,C 180,E1 -3771.846,E2 -3771.846} C_VEL
LIN {X 0,Y 545.154,Z 201.579,A -85,B 0,C 180,E1 -3774.822,E2 -3774.822} C_VEL
LIN {X 0,Y 545.134,Z 201.576,A -85,B 0,C 180,E1 -3777.783,E2 -3777.783} C_VEL
LIN {X 0,Y 545.166,Z 201.578,A -85,B 0,C 180,E1 -3780.738,E2 -3780.738} C_VEL
LIN {X 0,Y 545.127,Z 201.585,A -85,B 0,C 180,E1 -3782.956,E2 -3782.956} C_VEL
LIN {X 0,Y 545.125,Z 201.577,A -85,B 0,C 180,E1 -3785.92,E2 -3785.92} C_VEL
LIN {X 0,Y 545.08,Z 201.583,A -85,B 0,C 180,E1 -3788.153,E2 -3788.153} C_VEL
LIN {X 0,Y 545.103,Z 201.582,A -85,B 0,C 180,E1 -3791.151,E2 -3791.151} C_VEL
LIN {X 0,Y 545.046,Z 201.589,A -85,B 0,C 180,E1 -3794.181,E2 -3794.181} C_VEL
LIN {X 0,Y 545.09,Z 201.581,A -85,B 0,C 180,E1 -3797.447,E2 -3797.447} C_VEL
LIN {X 0,Y 545.057,Z 201.592,A -85,B 0,C 180,E1 -3800.373,E2 -3800.373} C_VEL
LIN {X 0,Y 545.05,Z 201.591,A -85,B 0,C 180,E1 -3802.757,E2 -3802.757} C_VEL
LIN {X 0,Y 545.054,Z 201.585,A -85,B 0,C 180,E1 -3805.513,E2 -3805.513} C_VEL
LIN {X 0,Y 545.075,Z 201.591,A -85,B 0,C 180,E1 -3808.494,E2 -3808.494} C_VEL
LIN {X 0,Y 545.027,Z 201.589,A -85,B 0,C 180,E1 -3811.05,E2 -3811.05} C_VEL
LIN {X 0,Y 545.032,Z 201.59,A -85,B 0,C 180,E1 -3813.839,E2 -3813.839} C_VEL
LIN {X 0,Y 545.04,Z 201.588,A -85,B 0,C 180,E1 -3816.93,E2 -3816.93} C_VEL
LIN {X 0,Y 545.025,Z 201.589,A -85,B 0,C 180,E1 -3817.054,E2 -3817.054} C_VEL
LIN {X 0,Y 544.324,Z 201.679,A -85,B 0,C 180,E1 -3817.67,E2 -3817.67} C_VEL
LIN {X 0,Y 541.482,Z 202.033,A -85,B 0,C 180,E1 -3818.671,E2 -3818.671} C_VEL
LIN {X 0,Y 539.111,Z 202.328,A -85,B 0,C 180,E1 -3819.477,E2 -3819.477} C_VEL
LIN {X 0,Y 538.104,Z 202.46,A -85,B 0,C 180,E1 -3820.099,E2 -3820.099} C_VEL
LIN {X 0,Y 538.027,Z 202.461,A -85,B 0,C 180,E1 -3820.31,E2 -3820.31} C_VEL
LIN {X 0,Y 538.001,Z 202.464,A -85,B 0,C 180,E1 -3822.992,E2 -3822.992} C_VEL
LIN {X 0,Y 537.999,Z 202.472,A -85,B 0,C 180,E1 -3825.928,E2 -3825.928} C_VEL
LIN {X 0,Y 538.052,Z 202.458,A -85,B 0,C 180,E1 -3829.252,E2 -3829.252} C_VEL
LIN {X 0,Y 537.971,Z 202.474,A -85,B 0,C 180,E1 -3832.126,E2 -3832.126} C_VEL
LIN {X 0,Y 538,Z 202.464,A -85,B 0,C 180,E1 -3834.92,E2 -3834.92} C_VEL
LIN {X 0,Y 538.014,Z 202.468,A -85,B 0,C 180,E1 -3837.621,E2 -3837.621} C_VEL
LIN {X 0,Y 538.027,Z 202.463,A -85,B 0,C 180,E1 -3840.243,E2 -3840.243} C_VEL
LIN {X 0,Y 538.058,Z 202.457,A -85,B 0,C 180,E1 -3842.799,E2 -3842.799} C_VEL
LIN {X 0,Y 538.039,Z 202.463,A -85,B 0,C 180,E1 -3845.295,E2 -3845.295} C_VEL
LIN {X 0,Y 538.006,Z 202.467,A -85,B 0,C 180,E1 -3848.044,E2 -3848.044} C_VEL
LIN {X 0,Y 538.029,Z 202.462,A -85,B 0,C 180,E1 -3850.942,E2 -3850.942} C_VEL
LIN {X 0,Y 538.019,Z 202.468,A -85,B 0,C 180,E1 -3853.301,E2 -3853.301} C_VEL
LIN {X 0,Y 538.059,Z 202.464,A -85,B 0,C 180,E1 -3855.632,E2 -3855.632} C_VEL
LIN {X 0,Y 538.075,Z 202.455,A -85,B 0,C 180,E1 -3858.703,E2 -3858.703} C_VEL
LIN {X 0,Y 538.084,Z 202.457,A -85,B 0,C 180,E1 -3861.741,E2 -3861.741} C_VEL
LIN {X 0,Y 538.161,Z 202.446,A -85,B 0,C 180,E1 -3864.756,E2 -3864.756} C_VEL
LIN {X 0,Y 538.169,Z 202.445,A -85,B 0,C 180,E1 -3867.755,E2 -3867.755} C_VEL
LIN {X 0,Y 538.18,Z 202.445,A -85,B 0,C 180,E1 -3870.748,E2 -3870.748} C_VEL
LIN {X 0,Y 538.136,Z 202.454,A -85,B 0,C 180,E1 -3872.994,E2 -3872.994} C_VEL
LIN {X 0,Y 538.119,Z 202.449,A -85,B 0,C 180,E1 -3875.997,E2 -3875.997} C_VEL
LIN {X 0,Y 538.067,Z 202.465,A -85,B 0,C 180,E1 -3879.017,E2 -3879.017} C_VEL
LIN {X 0,Y 538.08,Z 202.454,A -85,B 0,C 180,E1 -3882.061,E2 -3882.061} C_VEL
LIN {X 0,Y 538.041,Z 202.465,A -85,B 0,C 180,E1 -3885.142,E2 -3885.142} C_VEL
LIN {X 0,Y 538.028,Z 202.462,A -85,B 0,C 180,E1 -3888.268,E2 -3888.268} C_VEL
LIN {X 0,Y 538.035,Z 202.467,A -85,B 0,C 180,E1 -3890.649,E2 -3890.649} C_VEL
LIN {X 0,Y 538.014,Z 202.462,A -85,B 0,C 180,E1 -3893.885,E2 -3893.885} C_VEL
LIN {X 0,Y 538.039,Z 202.465,A -85,B 0,C 180,E1 -3896.364,E2 -3896.364} C_VEL
LIN {X 0,Y 538.042,Z 202.466,A -85,B 0,C 180,E1 -3898.936,E2 -3898.936} C_VEL
LIN {X 0,Y 538.101,Z 202.531,A -85,B 0,C 180,E1 -3901.272,E2 -3901.272} C_VEL
LIN {X 0,Y 538.385,Z 208.071,A -85,B 0,C 180,E1 -3902.354,E2 -3902.354} C_VEL
LIN {X 0,Y 538.184,Z 223.436,A -85,B 0,C 180,E1 -3905.309,E2 -3905.309} C_VEL
LIN {X 0,Y 539.68,Z 232.554,A -85,B 0,C 180,E1 -3905.483,E2 -3905.483} C_VEL
LIN {X 0,Y 539.239,Z 330.412,A -85,B 0,C 180,E1 -3906.818,E2 -3906.818} C_VEL
LIN {X 0,Y 539.077,Z 343.674,A -85,B 0,C 180,E1 -3907.156,E2 -3907.156} C_VEL
LIN {X 0,Y 538.963,Z 356.351,A -85,B 0,C 180,E1 -3907.64,E2 -3907.64} C_VEL
LIN {X 0,Y 538.732,Z 368.633,A -85,B 0,C 180,E1 -3908.278,E2 -3908.278} C_VEL
LIN {X 0,Y 538.48,Z 379.827,A -85,B 0,C 180,E1 -3909.026,E2 -3909.026} C_VEL
LIN {X 0,Y 538.274,Z 390.128,A -85,B 0,C 180,E1 -3909.891,E2 -3909.891} C_VEL
LIN {X 0,Y 538.062,Z 399.792,A -85,B 0,C 180,E1 -3910.893,E2 -3910.893} C_VEL
LIN {X 0,Y 537.882,Z 408.729,A -85,B 0,C 180,E1 -3912.051,E2 -3912.051} C_VEL
LIN {X 0,Y 537.735,Z 415.448,A -85,B 0,C 180,E1 -3913.13,E2 -3913.13} C_VEL
LIN {X 0,Y 537.638,Z 421.884,A -85,B 0,C 180,E1 -3914.437,E2 -3914.437} C_VEL
LIN {X 0,Y 537.587,Z 426.141,A -85,B 0,C 180,E1 -3915.563,E2 -3915.563} C_VEL
LIN {X 0,Y 537.525,Z 430.207,A -85,B 0,C 180,E1 -3917.063,E2 -3917.063} C_VEL
LIN {X 0,Y 537.504,Z 432.112,A -85,B 0,C 180,E1 -3918.177,E2 -3918.177} C_VEL
LIN {X 0,Y 537.472,Z 433.147,A -85,B 0,C 180,E1 -3919.317,E2 -3919.317} C_VEL
LIN {X 0,Y 537.451,Z 433.266,A -85,B 0,C 180,E1 -3920.483,E2 -3920.483} C_VEL
LIN {X 0,Y 537.44,Z 432.407,A -85,B 0,C 180,E1 -3921.676,E2 -3921.676} C_VEL
LIN {X 0,Y 537.508,Z 430.218,A -85,B 0,C 180,E1 -3923.026,E2 -3923.026} C_VEL
LIN {X 0,Y 537.578,Z 426.198,A -85,B 0,C 180,E1 -3924.515,E2 -3924.515} C_VEL
LIN {X 0,Y 537.586,Z 421.3,A -85,B 0,C 180,E1 -3925.796,E2 -3925.796} C_VEL
LIN {X 0,Y 537.752,Z 415.418,A -85,B 0,C 180,E1 -3926.97,E2 -3926.97} C_VEL
LIN {X 0,Y 537.866,Z 408.168,A -85,B 0,C 180,E1 -3928.128,E2 -3928.128} C_VEL
LIN {X 0,Y 538.059,Z 400.173,A -85,B 0,C 180,E1 -3929.158,E2 -3929.158} C_VEL
LIN {X 0,Y 538.27,Z 390.739,A -85,B 0,C 180,E1 -3930.147,E2 -3930.147} C_VEL
LIN {X 0,Y 538.43,Z 381.005,A -85,B 0,C 180,E1 -3930.979,E2 -3930.979} C_VEL
LIN {X 0,Y 538.699,Z 369.314,A -85,B 0,C 180,E1 -3931.776,E2 -3931.776} C_VEL
LIN {X 0,Y 538.953,Z 358.312,A -85,B 0,C 180,E1 -3932.361,E2 -3932.361} C_VEL
LIN {X 0,Y 539.141,Z 346.087,A -85,B 0,C 180,E1 -3932.855,E2 -3932.855} C_VEL
LIN {X 0,Y 539.237,Z 333.834,A -85,B 0,C 180,E1 -3933.201,E2 -3933.201} C_VEL
LIN {X 0,Y 539.337,Z 316.465,A -85,B 0,C 180,E1 -3933.48,E2 -3933.48} C_VEL
LIN {X 0,Y 539.656,Z 231.316,A -85,B 0,C 180,E1 -3934.625,E2 -3934.625} C_VEL
LIN {X 0,Y 538.157,Z 223.299,A -85,B 0,C 180,E1 -3934.782,E2 -3934.782} C_VEL
LIN {X 0,Y 538.225,Z 208.972,A -85,B 0,C 180,E1 -3937.344,E2 -3937.344} C_VEL
LIN {X 0,Y 538.054,Z 202.463,A -85,B 0,C 180,E1 -3938.51,E2 -3938.51} C_VEL
LIN {X 0,Y 537.994,Z 202.47,A -85,B 0,C 180,E1 -3940.939,E2 -3940.939} C_VEL
LIN {X 0,Y 538.007,Z 202.472,A -85,B 0,C 180,E1 -3943.299,E2 -3943.299} C_VEL
LIN {X 0,Y 537.988,Z 202.469,A -85,B 0,C 180,E1 -3946.4,E2 -3946.4} C_VEL
LIN {X 0,Y 538.055,Z 202.462,A -85,B 0,C 180,E1 -3948.701,E2 -3948.701} C_VEL
LIN {X 0,Y 538.038,Z 202.463,A -85,B 0,C 180,E1 -3951.739,E2 -3951.739} C_VEL
LIN {X 0,Y 538.078,Z 202.456,A -85,B 0,C 180,E1 -3954.002,E2 -3954.002} C_VEL
LIN {X 0,Y 538.093,Z 202.461,A -85,B 0,C 180,E1 -3957.006,E2 -3957.006} C_VEL
LIN {X 0,Y 538.11,Z 202.451,A -85,B 0,C 180,E1 -3960,E2 -3960} C_VEL
LIN {X 0,Y 538.091,Z 202.461,A -85,B 0,C 180,E1 -3962.995,E2 -3962.995} C_VEL
LIN {X 0,Y 538.065,Z 202.455,A -85,B 0,C 180,E1 -3965.998,E2 -3965.998} C_VEL
LIN {X 0,Y 538.023,Z 202.469,A -85,B 0,C 180,E1 -3969.019,E2 -3969.019} C_VEL
LIN {X 0,Y 538.03,Z 202.46,A -85,B 0,C 180,E1 -3972.064,E2 -3972.064} C_VEL
LIN {X 0,Y 537.994,Z 202.469,A -85,B 0,C 180,E1 -3975.146,E2 -3975.146} C_VEL
LIN {X 0,Y 538.043,Z 202.459,A -85,B 0,C 180,E1 -3977.554,E2 -3977.554} C_VEL
LIN {X 0,Y 537.994,Z 202.472,A -85,B 0,C 180,E1 -3980.653,E2 -3980.653} C_VEL
LIN {X 0,Y 537.995,Z 202.464,A -85,B 0,C 180,E1 -3983.889,E2 -3983.889} C_VEL
LIN {X 0,Y 538.004,Z 202.47,A -85,B 0,C 180,E1 -3986.369,E2 -3986.369} C_VEL
LIN {X 0,Y 537.993,Z 202.467,A -85,B 0,C 180,E1 -3988.937,E2 -3988.937} C_VEL
LIN {X 0,Y 537.987,Z 202.468,A -85,B 0,C 180,E1 -3991.893,E2 -3991.893} C_VEL
LIN {X 0,Y 537.992,Z 202.47,A -85,B 0,C 180,E1 -3994.624,E2 -3994.624} C_VEL
LIN {X 0,Y 537.974,Z 202.468,A -85,B 0,C 180,E1 -3997.174,E2 -3997.174} C_VEL
LIN {X 0,Y 537.993,Z 202.468,A -85,B 0,C 180,E1 -3999.8,E2 -3999.8} C_VEL
LIN {X 0,Y 537.99,Z 202.467,A -85,B 0,C 180,E1 -4002.789,E2 -4002.789} C_VEL
LIN {X 0,Y 537.981,Z 202.466,A -85,B 0,C 180,E1 -4005.141,E2 -4005.141} C_VEL
LIN {X 0,Y 538.017,Z 202.471,A -85,B 0,C 180,E1 -4008.231,E2 -4008.231} C_VEL
LIN {X 0,Y 537.992,Z 202.466,A -85,B 0,C 180,E1 -4011.173,E2 -4011.173} C_VEL
LIN {X 0,Y 538.009,Z 202.472,A -85,B 0,C 180,E1 -4014.087,E2 -4014.087} C_VEL
LIN {X 0,Y 538.015,Z 202.464,A -85,B 0,C 180,E1 -4016.73,E2 -4016.73} C_VEL
LIN {X 0,Y 538.014,Z 202.468,A -85,B 0,C 180,E1 -4019.559,E2 -4019.559} C_VEL
LIN {X 0,Y 538.028,Z 202.47,A -85,B 0,C 180,E1 -4021.953,E2 -4021.953} C_VEL
LIN {X 0,Y 538.063,Z 202.461,A -85,B 0,C 180,E1 -4024.47,E2 -4024.47} C_VEL
LIN {X 0,Y 538.062,Z 202.589,A -85,B 0,C 180,E1 -4025.566,E2 -4025.566} C_VEL
LIN {X 0,Y 539.156,Z 209.205,A -85,B 0,C 180,E1 -4026.576,E2 -4026.576} C_VEL
LIN {X 0,Y 538.92,Z 227.132,A -85,B 0,C 180,E1 -4029.187,E2 -4029.187} C_VEL
LIN {X 0,Y 538.558,Z 248.736,A -85,B 0,C 180,E1 -4032.294,E2 -4032.294} C_VEL
LIN {X 0,Y 538.262,Z 269.305,A -85,B 0,C 180,E1 -4035.217,E2 -4035.217} C_VEL
LIN {X 0,Y 538.785,Z 272.922,A -85,B 0,C 180,E1 -4035.308,E2 -4035.308} C_VEL
LIN {X 0,Y 539.594,Z 280.095,A -85,B 0,C 180,E1 -4035.429,E2 -4035.429} C_VEL
LIN {X 0,Y 539.239,Z 378.693,A -85,B 0,C 180,E1 -4036.769,E2 -4036.769} C_VEL
LIN {X 0,Y 539.054,Z 392.587,A -85,B 0,C 180,E1 -4037.124,E2 -4037.124} C_VEL
LIN {X 0,Y 538.839,Z 405.555,A -85,B 0,C 180,E1 -4037.621,E2 -4037.621} C_VEL
LIN {X 0,Y 538.658,Z 417.71,A -85,B 0,C 180,E1 -4038.259,E2 -4038.259} C_VEL
LIN {X 0,Y 538.44,Z 428.766,A -85,B 0,C 180,E1 -4038.996,E2 -4038.996} C_VEL
LIN {X 0,Y 538.218,Z 439.042,A -85,B 0,C 180,E1 -4039.848,E2 -4039.848} C_VEL
LIN {X 0,Y 537.997,Z 448.275,A -85,B 0,C 180,E1 -4040.793,E2 -4040.793} C_VEL
LIN {X 0,Y 537.824,Z 457.27,A -85,B 0,C 180,E1 -4041.925,E2 -4041.925} C_VEL
LIN {X 0,Y 537.69,Z 464.511,A -85,B 0,C 180,E1 -4043.056,E2 -4043.056} C_VEL
LIN {X 0,Y 537.656,Z 471.105,A -85,B 0,C 180,E1 -4044.374,E2 -4044.374} C_VEL
LIN {X 0,Y 537.554,Z 475.461,A -85,B 0,C 180,E1 -4045.501,E2 -4045.501} C_VEL
LIN {X 0,Y 537.591,Z 477.771,A -85,B 0,C 180,E1 -4046.253,E2 -4046.253} C_VEL
LIN {X 0,Y 537.551,Z 479.64,A -85,B 0,C 180,E1 -4047.003,E2 -4047.003} C_VEL
LIN {X 0,Y 537.49,Z 481.039,A -85,B 0,C 180,E1 -4047.752,E2 -4047.752} C_VEL
LIN {X 0,Y 537.443,Z 482.649,A -85,B 0,C 180,E1 -4049.251,E2 -4049.251} C_VEL
LIN {X 0,Y 537.443,Z 482.867,A -85,B 0,C 180,E1 -4050,E2 -4050} C_VEL
LIN {X 0,Y 537.443,Z 482.65,A -85,B 0,C 180,E1 -4050.749,E2 -4050.749} C_VEL
LIN {X 0,Y 537.49,Z 481.046,A -85,B 0,C 180,E1 -4052.248,E2 -4052.248} C_VEL
LIN {X 0,Y 537.551,Z 479.648,A -85,B 0,C 180,E1 -4052.997,E2 -4052.997} C_VEL
LIN {X 0,Y 537.603,Z 476.704,A -85,B 0,C 180,E1 -4054.123,E2 -4054.123} C_VEL
LIN {X 0,Y 537.587,Z 472.714,A -85,B 0,C 180,E1 -4055.25,E2 -4055.25} C_VEL
LIN {X 0,Y 537.633,Z 467.844,A -85,B 0,C 180,E1 -4056.325,E2 -4056.325} C_VEL
LIN {X 0,Y 537.75,Z 461.117,A -85,B 0,C 180,E1 -4057.509,E2 -4057.509} C_VEL
LIN {X 0,Y 537.92,Z 453.054,A -85,B 0,C 180,E1 -4058.64,E2 -4058.64} C_VEL
LIN {X 0,Y 538.089,Z 444.836,A -85,B 0,C 180,E1 -4059.585,E2 -4059.585} C_VEL
LIN {X 0,Y 538.342,Z 434.815,A -85,B 0,C 180,E1 -4060.53,E2 -4060.53} C_VEL
LIN {X 0,Y 538.505,Z 424.916,A -85,B 0,C 180,E1 -4061.288,E2 -4061.288} C_VEL
LIN {X 0,Y 538.728,Z 413.734,A -85,B 0,C 180,E1 -4061.974,E2 -4061.974} C_VEL
LIN {X 0,Y 538.919,Z 401.212,A -85,B 0,C 180,E1 -4062.568,E2 -4062.568} C_VEL
LIN {X 0,Y 539.158,Z 388.89,A -85,B 0,C 180,E1 -4062.993,E2 -4062.993} C_VEL
LIN {X 0,Y 539.279,Z 376.236,A -85,B 0,C 180,E1 -4063.277,E2 -4063.277} C_VEL
LIN {X 0,Y 539.49,Z 277.641,A -85,B 0,C 180,E1 -4064.61,E2 -4064.61} C_VEL
LIN {X 0,Y 538.331,Z 269.732,A -85,B 0,C 180,E1 -4064.76,E2 -4064.76} C_VEL
LIN {X 0,Y 538.606,Z 249.23,A -85,B 0,C 180,E1 -4067.722,E2 -4067.722} C_VEL
LIN {X 0,Y 538.993,Z 229.404,A -85,B 0,C 180,E1 -4070.611,E2 -4070.611} C_VEL
LIN {X 0,Y 539.425,Z 210.54,A -85,B 0,C 180,E1 -4073.411,E2 -4073.411} C_VEL
LIN {X 0,Y 538.073,Z 202.462,A -85,B 0,C 180,E1 -4074.703,E2 -4074.703} C_VEL
LIN {X 0,Y 538.038,Z 202.463,A -85,B 0,C 180,E1 -4077.347,E2 -4077.347} C_VEL
LIN {X 0,Y 538.006,Z 202.47,A -85,B 0,C 180,E1 -4079.758,E2 -4079.758} C_VEL
LIN {X 0,Y 538.004,Z 202.468,A -85,B 0,C 180,E1 -4082.38,E2 -4082.38} C_VEL
LIN {X 0,Y 537.996,Z 202.465,A -85,B 0,C 180,E1 -4085.08,E2 -4085.08} C_VEL
LIN {X 0,Y 537.973,Z 202.476,A -85,B 0,C 180,E1 -4087.874,E2 -4087.874} C_VEL
LIN {X 0,Y 538.028,Z 202.461,A -85,B 0,C 180,E1 -4090.772,E2 -4090.772} C_VEL
LIN {X 0,Y 537.998,Z 202.47,A -85,B 0,C 180,E1 -4094.071,E2 -4094.071} C_VEL
LIN {X 0,Y 537.994,Z 202.467,A -85,B 0,C 180,E1 -4097.211,E2 -4097.211} C_VEL
LIN {X 0,Y 538.002,Z 202.466,A -85,B 0,C 180,E1 -4100.201,E2 -4100.201} C_VEL
LIN {X 0,Y 537.996,Z 202.466,A -85,B 0,C 180,E1 -4103.064,E2 -4103.064} C_VEL
LIN {X 0,Y 537.993,Z 202.471,A -85,B 0,C 180,E1 -4105.825,E2 -4105.825} C_VEL
LIN {X 0,Y 537.982,Z 202.466,A -85,B 0,C 180,E1 -4108.497,E2 -4108.497} C_VEL
LIN {X 0,Y 538.016,Z 202.466,A -85,B 0,C 180,E1 -4111.097,E2 -4111.097} C_VEL
LIN {X 0,Y 538.003,Z 202.47,A -85,B 0,C 180,E1 -4113.631,E2 -4113.631} C_VEL
LIN {X 0,Y 537.994,Z 202.466,A -85,B 0,C 180,E1 -4116.111,E2 -4116.111} C_VEL
LIN {X 0,Y 537.993,Z 202.474,A -85,B 0,C 180,E1 -4119.347,E2 -4119.347} C_VEL
LIN {X 0,Y 538.04,Z 202.46,A -85,B 0,C 180,E1 -4122.516,E2 -4122.516} C_VEL
LIN {X 0,Y 538.009,Z 202.466,A -85,B 0,C 180,E1 -4125.629,E2 -4125.629} C_VEL
LIN {X 0,Y 538.053,Z 202.46,A -85,B 0,C 180,E1 -4128.701,E2 -4128.701} C_VEL
LIN {X 0,Y 538.035,Z 202.461,A -85,B 0,C 180,E1 -4131.739,E2 -4131.739} C_VEL
LIN {X 0,Y 538.11,Z 202.455,A -85,B 0,C 180,E1 -4134.754,E2 -4134.754} C_VEL
LIN {X 0,Y 538.107,Z 202.451,A -85,B 0,C 180,E1 -4137.754,E2 -4137.754} C_VEL
LIN {X 0,Y 538.135,Z 202.454,A -85,B 0,C 180,E1 -4140.748,E2 -4140.748} C_VEL
LIN {X 0,Y 538.092,Z 202.46,A -85,B 0,C 180,E1 -4142.994,E2 -4142.994} C_VEL
LIN {X 0,Y 538.077,Z 202.455,A -85,B 0,C 180,E1 -4145.998,E2 -4145.998} C_VEL
LIN {X 0,Y 538.037,Z 202.462,A -85,B 0,C 180,E1 -4148.261,E2 -4148.261} C_VEL
LIN {X 0,Y 538.049,Z 202.458,A -85,B 0,C 180,E1 -4151.61,E2 -4151.61} C_VEL
LIN {X 0,Y 538.003,Z 202.47,A -85,B 0,C 180,E1 -4154.858,E2 -4154.858} C_VEL
LIN {X 0,Y 538.04,Z 202.459,A -85,B 0,C 180,E1 -4157.554,E2 -4157.554} C_VEL
LIN {X 0,Y 538.004,Z 202.471,A -85,B 0,C 180,E1 -4160.652,E2 -4160.652} C_VEL
LIN {X 0,Y 538.022,Z 202.463,A -85,B 0,C 180,E1 -4163.071,E2 -4163.071} C_VEL
LIN {X 0,Y 538.003,Z 202.464,A -85,B 0,C 180,E1 -4165.677,E2 -4165.677} C_VEL
LIN {X 0,Y 538.012,Z 202.467,A -85,B 0,C 180,E1 -4168.051,E2 -4168.051} C_VEL
LIN {X 0,Y 537.984,Z 202.471,A -85,B 0,C 180,E1 -4170.629,E2 -4170.629} C_VEL
LIN {X 0,Y 538.002,Z 202.464,A -85,B 0,C 180,E1 -4173.286,E2 -4173.286} C_VEL
LIN {X 0,Y 537.989,Z 202.471,A -85,B 0,C 180,E1 -4176.005,E2 -4176.005} C_VEL
LIN {X 0,Y 537.984,Z 202.467,A -85,B 0,C 180,E1 -4178.833,E2 -4178.833} C_VEL
LIN {X 0,Y 538.027,Z 202.461,A -85,B 0,C 180,E1 -4180.31,E2 -4180.31} C_VEL
LIN {X 0,Y 537.368,Z 202.545,A -85,B 0,C 180,E1 -4180.935,E2 -4180.935} C_VEL
LIN {X 0,Y 534.501,Z 202.906,A -85,B 0,C 180,E1 -4181.95,E2 -4181.95} C_VEL
LIN {X 0,Y 532.068,Z 203.208,A -85,B 0,C 180,E1 -4182.766,E2 -4182.766} C_VEL
LIN {X 0,Y 531.018,Z 203.336,A -85,B 0,C 180,E1 -4183.397,E2 -4183.397} C_VEL
LIN {X 0,Y 530.93,Z 203.346,A -85,B 0,C 180,E1 -4183.611,E2 -4183.611} C_VEL
LIN {X 0,Y 530.934,Z 203.347,A -85,B 0,C 180,E1 -4186.508,E2 -4186.508} C_VEL
LIN {X 0,Y 531.001,Z 203.339,A -85,B 0,C 180,E1 -4189.574,E2 -4189.574} C_VEL
LIN {X 0,Y 530.946,Z 203.344,A -85,B 0,C 180,E1 -4192.58,E2 -4192.58} C_VEL
LIN {X 0,Y 530.983,Z 203.34,A -85,B 0,C 180,E1 -4195.314,E2 -4195.314} C_VEL
LIN {X 0,Y 530.965,Z 203.346,A -85,B 0,C 180,E1 -4198.036,E2 -4198.036} C_VEL
LIN {X 0,Y 530.981,Z 203.339,A -85,B 0,C 180,E1 -4200.875,E2 -4200.875} C_VEL
LIN {X 0,Y 530.999,Z 203.339,A -85,B 0,C 180,E1 -4203.259,E2 -4203.259} C_VEL
LIN {X 0,Y 530.986,Z 203.343,A -85,B 0,C 180,E1 -4205.96,E2 -4205.96} C_VEL
LIN {X 0,Y 530.991,Z 203.339,A -85,B 0,C 180,E1 -4209.064,E2 -4209.064} C_VEL
LIN {X 0,Y 531.01,Z 203.335,A -85,B 0,C 180,E1 -4212.28,E2 -4212.28} C_VEL
LIN {X 0,Y 531.036,Z 203.34,A -85,B 0,C 180,E1 -4215.438,E2 -4215.438} C_VEL
LIN {X 0,Y 531.034,Z 203.332,A -85,B 0,C 180,E1 -4218.551,E2 -4218.551} C_VEL
LIN {X 0,Y 531.053,Z 203.335,A -85,B 0,C 180,E1 -4221.63,E2 -4221.63} C_VEL
LIN {X 0,Y 531.12,Z 203.323,A -85,B 0,C 180,E1 -4224.686,E2 -4224.686} C_VEL
LIN {X 0,Y 531.141,Z 203.321,A -85,B 0,C 180,E1 -4227.725,E2 -4227.725} C_VEL
LIN {X 0,Y 531.15,Z 203.32,A -85,B 0,C 180,E1 -4230.758,E2 -4230.758} C_VEL
LIN {X 0,Y 531.103,Z 203.331,A -85,B 0,C 180,E1 -4233.034,E2 -4233.034} C_VEL
LIN {X 0,Y 531.072,Z 203.327,A -85,B 0,C 180,E1 -4236.077,E2 -4236.077} C_VEL
LIN {X 0,Y 531.054,Z 203.33,A -85,B 0,C 180,E1 -4238.37,E2 -4238.37} C_VEL
LIN {X 0,Y 531.048,Z 203.331,A -85,B 0,C 180,E1 -4241.671,E2 -4241.671} C_VEL
LIN {X 0,Y 531.026,Z 203.342,A -85,B 0,C 180,E1 -4244.954,E2 -4244.954} C_VEL
LIN {X 0,Y 531.011,Z 203.335,A -85,B 0,C 180,E1 -4247.721,E2 -4247.721} C_VEL
LIN {X 0,Y 530.994,Z 203.344,A -85,B 0,C 180,E1 -4250.936,E2 -4250.936} C_VEL
LIN {X 0,Y 530.97,Z 203.342,A -85,B 0,C 180,E1 -4254.222,E2 -4254.222} C_VEL
LIN {X 0,Y 531.001,Z 203.345,A -85,B 0,C 180,E1 -4256.741,E2 -4256.741} C_VEL
LIN {X 0,Y 530.986,Z 203.342,A -85,B 0,C 180,E1 -4259.319,E2 -4259.319} C_VEL
LIN {X 0,Y 531.063,Z 203.466,A -85,B 0,C 180,E1 -4261.179,E2 -4261.179} C_VEL
LIN {X 0,Y 531.406,Z 208.497,A -85,B 0,C 180,E1 -4262.176,E2 -4262.176} C_VEL
LIN {X 0,Y 531.213,Z 223.607,A -85,B 0,C 180,E1 -4265.098,E2 -4265.098} C_VEL
LIN {X 0,Y 532.814,Z 233.512,A -85,B 0,C 180,E1 -4265.302,E2 -4265.302} C_VEL
LIN {X 0,Y 532.331,Z 330.769,A -85,B 0,C 180,E1 -4266.65,E2 -4266.65} C_VEL
LIN {X 0,Y 532.158,Z 343.902,A -85,B 0,C 180,E1 -4266.989,E2 -4266.989} C_VEL
LIN {X 0,Y 532.035,Z 356.78,A -85,B 0,C 180,E1 -4267.488,E2 -4267.488} C_VEL
LIN {X 0,Y 531.792,Z 367.807,A -85,B 0,C 180,E1 -4268.06,E2 -4268.06} C_VEL
LIN {X 0,Y 531.545,Z 379.339,A -85,B 0,C 180,E1 -4268.827,E2 -4268.827} C_VEL
LIN {X 0,Y 531.295,Z 389.242,A -85,B 0,C 180,E1 -4269.648,E2 -4269.648} C_VEL
LIN {X 0,Y 531.053,Z 399.597,A -85,B 0,C 180,E1 -4270.717,E2 -4270.717} C_VEL
LIN {X 0,Y 530.87,Z 407.938,A -85,B 0,C 180,E1 -4271.788,E2 -4271.788} C_VEL
LIN {X 0,Y 530.683,Z 414.751,A -85,B 0,C 180,E1 -4272.861,E2 -4272.861} C_VEL
LIN {X 0,Y 530.604,Z 420.256,A -85,B 0,C 180,E1 -4273.928,E2 -4273.928} C_VEL
LIN {X 0,Y 530.533,Z 424.687,A -85,B 0,C 180,E1 -4274.996,E2 -4274.996} C_VEL
LIN {X 0,Y 530.464,Z 429.211,A -85,B 0,C 180,E1 -4276.454,E2 -4276.454} C_VEL
LIN {X 0,Y 530.403,Z 432.073,A -85,B 0,C 180,E1 -4277.896,E2 -4277.896} C_VEL
LIN {X 0,Y 530.401,Z 433.311,A -85,B 0,C 180,E1 -4279.042,E2 -4279.042} C_VEL
LIN {X 0,Y 530.371,Z 433.59,A -85,B 0,C 180,E1 -4280.502,E2 -4280.502} C_VEL
LIN {X 0,Y 530.346,Z 432.96,A -85,B 0,C 180,E1 -4281.477,E2 -4281.477} C_VEL
LIN {X 0,Y 530.393,Z 431.339,A -85,B 0,C 180,E1 -4282.65,E2 -4282.65} C_VEL
LIN {X 0,Y 530.484,Z 428.507,A -85,B 0,C 180,E1 -4283.906,E2 -4283.906} C_VEL
LIN {X 0,Y 530.486,Z 424.067,A -85,B 0,C 180,E1 -4285.273,E2 -4285.273} C_VEL
LIN {X 0,Y 530.666,Z 418.483,A -85,B 0,C 180,E1 -4286.539,E2 -4286.539} C_VEL
LIN {X 0,Y 530.764,Z 411.545,A -85,B 0,C 180,E1 -4287.771,E2 -4287.771} C_VEL
LIN {X 0,Y 530.992,Z 403.379,A -85,B 0,C 180,E1 -4288.923,E2 -4288.923} C_VEL
LIN {X 0,Y 531.222,Z 393.507,A -85,B 0,C 180,E1 -4290.038,E2 -4290.038} C_VEL
LIN {X 0,Y 531.403,Z 383.327,A -85,B 0,C 180,E1 -4290.96,E2 -4290.96} C_VEL
LIN {X 0,Y 531.688,Z 371.784,A -85,B 0,C 180,E1 -4291.793,E2 -4291.793} C_VEL
LIN {X 0,Y 531.984,Z 359.873,A -85,B 0,C 180,E1 -4292.459,E2 -4292.459} C_VEL
LIN {X 0,Y 532.188,Z 348.336,A -85,B 0,C 180,E1 -4292.95,E2 -4292.95} C_VEL
LIN {X 0,Y 532.307,Z 335.135,A -85,B 0,C 180,E1 -4293.347,E2 -4293.347} C_VEL
LIN {X 0,Y 532.404,Z 319.699,A -85,B 0,C 180,E1 -4293.612,E2 -4293.612} C_VEL
LIN {X 0,Y 532.695,Z 231.74,A -85,B 0,C 180,E1 -4294.819,E2 -4294.819} C_VEL
LIN {X 0,Y 531.162,Z 223.419,A -85,B 0,C 180,E1 -4295.003,E2 -4295.003} C_VEL
LIN {X 0,Y 531.219,Z 208.327,A -85,B 0,C 180,E1 -4297.684,E2 -4297.684} C_VEL
LIN {X 0,Y 531.013,Z 203.341,A -85,B 0,C 180,E1 -4298.58,E2 -4298.58} C_VEL
LIN {X 0,Y 530.951,Z 203.352,A -85,B 0,C 180,E1 -4301.478,E2 -4301.478} C_VEL
LIN {X 0,Y 530.959,Z 203.346,A -85,B 0,C 180,E1 -4303.862,E2 -4303.862} C_VEL
LIN {X 0,Y 530.941,Z 203.347,A -85,B 0,C 180,E1 -4306.216,E2 -4306.216} C_VEL
LIN {X 0,Y 531.006,Z 203.339,A -85,B 0,C 180,E1 -4308.549,E2 -4308.549} C_VEL
LIN {X 0,Y 531.007,Z 203.34,A -85,B 0,C 180,E1 -4311.629,E2 -4311.629} C_VEL
LIN {X 0,Y 531.036,Z 203.333,A -85,B 0,C 180,E1 -4313.923,E2 -4313.923} C_VEL
LIN {X 0,Y 531.059,Z 203.336,A -85,B 0,C 180,E1 -4316.966,E2 -4316.966} C_VEL
LIN {X 0,Y 531.081,Z 203.327,A -85,B 0,C 180,E1 -4320,E2 -4320} C_VEL
LIN {X 0,Y 531.057,Z 203.337,A -85,B 0,C 180,E1 -4323.035,E2 -4323.035} C_VEL
LIN {X 0,Y 531.02,Z 203.333,A -85,B 0,C 180,E1 -4326.078,E2 -4326.078} C_VEL
LIN {X 0,Y 530.983,Z 203.344,A -85,B 0,C 180,E1 -4329.139,E2 -4329.139} C_VEL
LIN {X 0,Y 531.013,Z 203.334,A -85,B 0,C 180,E1 -4331.681,E2 -4331.681} C_VEL
LIN {X 0,Y 530.977,Z 203.346,A -85,B 0,C 180,E1 -4334.957,E2 -4334.957} C_VEL
LIN {X 0,Y 530.979,Z 203.338,A -85,B 0,C 180,E1 -4337.724,E2 -4337.724} C_VEL
LIN {X 0,Y 530.956,Z 203.347,A -85,B 0,C 180,E1 -4340.94,E2 -4340.94} C_VEL
LIN {X 0,Y 530.961,Z 203.341,A -85,B 0,C 180,E1 -4344.047,E2 -4344.047} C_VEL
LIN {X 0,Y 530.966,Z 203.347,A -85,B 0,C 180,E1 -4346.746,E2 -4346.746} C_VEL
LIN {X 0,Y 530.942,Z 203.343,A -85,B 0,C 180,E1 -4349.325,E2 -4349.325} C_VEL
LIN {X 0,Y 530.94,Z 203.348,A -85,B 0,C 180,E1 -4352.106,E2 -4352.106} C_VEL
LIN {X 0,Y 530.95,Z 203.344,A -85,B 0,C 180,E1 -4354.857,E2 -4354.857} C_VEL
LIN {X 0,Y 530.932,Z 203.345,A -85,B 0,C 180,E1 -4357.511,E2 -4357.511} C_VEL
LIN {X 0,Y 530.952,Z 203.349,A -85,B 0,C 180,E1 -4360.436,E2 -4360.436} C_VEL
LIN {X 0,Y 530.937,Z 203.343,A -85,B 0,C 180,E1 -4363.285,E2 -4363.285} C_VEL
LIN {X 0,Y 530.952,Z 203.344,A -85,B 0,C 180,E1 -4365.625,E2 -4365.625} C_VEL
LIN {X 0,Y 530.977,Z 203.343,A -85,B 0,C 180,E1 -4368.568,E2 -4368.568} C_VEL
LIN {X 0,Y 530.936,Z 203.347,A -85,B 0,C 180,E1 -4371.533,E2 -4371.533} C_VEL
LIN {X 0,Y 530.961,Z 203.346,A -85,B 0,C 180,E1 -4374.385,E2 -4374.385} C_VEL
LIN {X 0,Y 530.952,Z 203.344,A -85,B 0,C 180,E1 -4377.136,E2 -4377.136} C_VEL
LIN {X 0,Y 530.958,Z 203.35,A -85,B 0,C 180,E1 -4379.806,E2 -4379.806} C_VEL
LIN {X 0,Y 531.001,Z 203.34,A -85,B 0,C 180,E1 -4382.471,E2 -4382.471} C_VEL
LIN {X 0,Y 531.034,Z 203.417,A -85,B 0,C 180,E1 -4385.417,E2 -4385.417} C_VEL
LIN {X 0,Y 532.194,Z 210.135,A -85,B 0,C 180,E1 -4386.458,E2 -4386.458} C_VEL
LIN {X 0,Y 531.986,Z 226.739,A -85,B 0,C 180,E1 -4388.902,E2 -4388.902} C_VEL
LIN {X 0,Y 531.551,Z 249.166,A -85,B 0,C 180,E1 -4392.169,E2 -4392.169} C_VEL
LIN {X 0,Y 531.252,Z 269.076,A -85,B 0,C 180,E1 -4395.038,E2 -4395.038} C_VEL
LIN {X 0,Y 532.716,Z 279.684,A -85,B 0,C 180,E1 -4395.236,E2 -4395.236} C_VEL
LIN {X 0,Y 532.339,Z 378.036,A -85,B 0,C 180,E1 -4396.595,E2 -4396.595} C_VEL
LIN {X 0,Y 532.15,Z 391.261,A -85,B 0,C 180,E1 -4396.93,E2 -4396.93} C_VEL
LIN {X 0,Y 531.909,Z 403.991,A -85,B 0,C 180,E1 -4397.409,E2 -4397.409} C_VEL
LIN {X 0,Y 531.708,Z 416.08,A -85,B 0,C 180,E1 -4398.032,E2 -4398.032} C_VEL
LIN {X 0,Y 531.43,Z 428.329,A -85,B 0,C 180,E1 -4398.849,E2 -4398.849} C_VEL
LIN {X 0,Y 531.141,Z 438.625,A -85,B 0,C 180,E1 -4399.711,E2 -4399.711} C_VEL
LIN {X 0,Y 530.949,Z 447.879,A -85,B 0,C 180,E1 -4400.669,E2 -4400.669} C_VEL
LIN {X 0,Y 530.76,Z 456.888,A -85,B 0,C 180,E1 -4401.817,E2 -4401.817} C_VEL
LIN {X 0,Y 530.626,Z 464.144,A -85,B 0,C 180,E1 -4402.964,E2 -4402.964} C_VEL
LIN {X 0,Y 530.572,Z 470.749,A -85,B 0,C 180,E1 -4404.299,E2 -4404.299} C_VEL
LIN {X 0,Y 530.452,Z 475.114,A -85,B 0,C 180,E1 -4405.441,E2 -4405.441} C_VEL
LIN {X 0,Y 530.516,Z 477.428,A -85,B 0,C 180,E1 -4406.202,E2 -4406.202} C_VEL
LIN {X 0,Y 530.457,Z 479.303,A -85,B 0,C 180,E1 -4406.962,E2 -4406.962} C_VEL
LIN {X 0,Y 530.411,Z 480.706,A -85,B 0,C 180,E1 -4407.722,E2 -4407.722} C_VEL
LIN {X 0,Y 530.35,Z 482.32,A -85,B 0,C 180,E1 -4409.241,E2 -4409.241} C_VEL
LIN {X 0,Y 530.351,Z 482.54,A -85,B 0,C 180,E1 -4410,E2 -4410} C_VEL
LIN {X 0,Y 530.361,Z 481.716,A -85,B 0,C 180,E1 -4411.518,E2 -4411.518} C_VEL
LIN {X 0,Y 530.411,Z 480.72,A -85,B 0,C 180,E1 -4412.278,E2 -4412.278} C_VEL
LIN {X 0,Y 530.457,Z 479.321,A -85,B 0,C 180,E1 -4413.037,E2 -4413.037} C_VEL
LIN {X 0,Y 530.522,Z 476.375,A -85,B 0,C 180,E1 -4414.178,E2 -4414.178} C_VEL
LIN {X 0,Y 530.521,Z 472.382,A -85,B 0,C 180,E1 -4415.32,E2 -4415.32} C_VEL
LIN {X 0,Y 530.59,Z 466.672,A -85,B 0,C 180,E1 -4416.573,E2 -4416.573} C_VEL
LIN {X 0,Y 530.719,Z 459.527,A -85,B 0,C 180,E1 -4417.8,E2 -4417.8} C_VEL
LIN {X 0,Y 530.895,Z 451.199,A -85,B 0,C 180,E1 -4418.947,E2 -4418.947} C_VEL
LIN {X 0,Y 531.066,Z 442.653,A -85,B 0,C 180,E1 -4419.905,E2 -4419.905} C_VEL
LIN {X 0,Y 531.325,Z 432.097,A -85,B 0,C 180,E1 -4420.863,E2 -4420.863} C_VEL
LIN {X 0,Y 531.603,Z 421.199,A -85,B 0,C 180,E1 -4421.66,E2 -4421.66} C_VEL
LIN {X 0,Y 531.819,Z 410.188,A -85,B 0,C 180,E1 -4422.302,E2 -4422.302} C_VEL
LIN {X 0,Y 532.035,Z 398.359,A -85,B 0,C 180,E1 -4422.83,E2 -4422.83} C_VEL
LIN {X 0,Y 532.251,Z 384.725,A -85,B 0,C 180,E1 -4423.262,E2 -4423.262} C_VEL
LIN {X 0,Y 532.423,Z 372.591,A -85,B 0,C 180,E1 -4423.5,E2 -4423.5} C_VEL
LIN {X 0,Y 532.62,Z 278.437,A -85,B 0,C 180,E1 -4424.787,E2 -4424.787} C_VEL
LIN {X 0,Y 531.304,Z 269.409,A -85,B 0,C 180,E1 -4424.963,E2 -4424.963} C_VEL
LIN {X 0,Y 531.655,Z 247.951,A -85,B 0,C 180,E1 -4428.111,E2 -4428.111} C_VEL
LIN {X 0,Y 532.114,Z 227.778,A -85,B 0,C 180,E1 -4431.092,E2 -4431.092} C_VEL
LIN {X 0,Y 532.498,Z 211.646,A -85,B 0,C 180,E1 -4433.528,E2 -4433.528} C_VEL
LIN {X 0,Y 531.028,Z 203.338,A -85,B 0,C 180,E1 -4434.896,E2 -4434.896} C_VEL
LIN {X 0,Y 531.002,Z 203.341,A -85,B 0,C 180,E1 -4437.593,E2 -4437.593} C_VEL
LIN {X 0,Y 530.961,Z 203.344,A -85,B 0,C 180,E1 -4440.642,E2 -4440.642} C_VEL
LIN {X 0,Y 530.973,Z 203.345,A -85,B 0,C 180,E1 -4443.769,E2 -4443.769} C_VEL
LIN {X 0,Y 530.948,Z 203.344,A -85,B 0,C 180,E1 -4446.554,E2 -4446.554} C_VEL
LIN {X 0,Y 530.959,Z 203.35,A -85,B 0,C 180,E1 -4449.851,E2 -4449.851} C_VEL
LIN {X 0,Y 530.956,Z 203.343,A -85,B 0,C 180,E1 -4452.453,E2 -4452.453} C_VEL
LIN {X 0,Y 530.958,Z 203.348,A -85,B 0,C 180,E1 -4455.618,E2 -4455.618} C_VEL
LIN {X 0,Y 530.969,Z 203.34,A -85,B 0,C 180,E1 -4458.562,E2 -4458.562} C_VEL
LIN {X 0,Y 530.922,Z 203.353,A -85,B 0,C 180,E1 -4461.526,E2 -4461.526} C_VEL
LIN {X 0,Y 530.945,Z 203.343,A -85,B 0,C 180,E1 -4464.379,E2 -4464.379} C_VEL
LIN {X 0,Y 530.935,Z 203.347,A -85,B 0,C 180,E1 -4467.131,E2 -4467.131} C_VEL
LIN {X 0,Y 530.927,Z 203.35,A -85,B 0,C 180,E1 -4469.8,E2 -4469.8} C_VEL
LIN {X 0,Y 530.973,Z 203.339,A -85,B 0,C 180,E1 -4472.463,E2 -4472.463} C_VEL
LIN {X 0,Y 530.961,Z 203.344,A -85,B 0,C 180,E1 -4474.94,E2 -4474.94} C_VEL
LIN {X 0,Y 530.942,Z 203.345,A -85,B 0,C 180,E1 -4477.892,E2 -4477.892} C_VEL
LIN {X 0,Y 530.947,Z 203.344,A -85,B 0,C 180,E1 -4480.675,E2 -4480.675} C_VEL
LIN {X 0,Y 530.965,Z 203.347,A -85,B 0,C 180,E1 -4483.07,E2 -4483.07} C_VEL
LIN {X 0,Y 530.964,Z 203.346,A -85,B 0,C 180,E1 -4485.434,E2 -4485.434} C_VEL
LIN {X 0,Y 531.005,Z 203.337,A -85,B 0,C 180,E1 -4488.549,E2 -4488.549} C_VEL
LIN {X 0,Y 531.004,Z 203.338,A -85,B 0,C 180,E1 -4491.628,E2 -4491.628} C_VEL
LIN {X 0,Y 531.068,Z 203.332,A -85,B 0,C 180,E1 -4494.684,E2 -4494.684} C_VEL
LIN {X 0,Y 531.079,Z 203.327,A -85,B 0,C 180,E1 -4497.724,E2 -4497.724} C_VEL
LIN {X 0,Y 531.104,Z 203.33,A -85,B 0,C 180,E1 -4500.758,E2 -4500.758} C_VEL
LIN {X 0,Y 531.058,Z 203.336,A -85,B 0,C 180,E1 -4503.034,E2 -4503.034} C_VEL
LIN {X 0,Y 531.035,Z 203.332,A -85,B 0,C 180,E1 -4506.077,E2 -4506.077} C_VEL
LIN {X 0,Y 531.006,Z 203.339,A -85,B 0,C 180,E1 -4508.371,E2 -4508.371} C_VEL
LIN {X 0,Y 531.011,Z 203.335,A -85,B 0,C 180,E1 -4511.682,E2 -4511.682} C_VEL
LIN {X 0,Y 530.975,Z 203.344,A -85,B 0,C 180,E1 -4514.957,E2 -4514.957} C_VEL
LIN {X 0,Y 530.977,Z 203.339,A -85,B 0,C 180,E1 -4517.723,E2 -4517.723} C_VEL
LIN {X 0,Y 530.973,Z 203.343,A -85,B 0,C 180,E1 -4520.939,E2 -4520.939} C_VEL
LIN {X 0,Y 530.96,Z 203.341,A -85,B 0,C 180,E1 -4523.396,E2 -4523.396} C_VEL
LIN {X 0,Y 530.968,Z 203.342,A -85,B 0,C 180,E1 -4525.899,E2 -4525.899} C_VEL
LIN {X 0,Y 530.959,Z 203.35,A -85,B 0,C 180,E1 -4528.458,E2 -4528.458} C_VEL
LIN {X 0,Y 530.924,Z 203.346,A -85,B 0,C 180,E1 -4531.081,E2 -4531.081} C_VEL
LIN {X 0,Y 530.952,Z 203.344,A -85,B 0,C 180,E1 -4533.775,E2 -4533.775} C_VEL
LIN {X 0,Y 530.932,Z 203.349,A -85,B 0,C 180,E1 -4536.56,E2 -4536.56} C_VEL
LIN {X 0,Y 531.009,Z 203.34,A -85,B 0,C 180,E1 -4539.865,E2 -4539.865} C_VEL
LIN {X 0,Y 530.955,Z 203.346,A -85,B 0,C 180,E1 -4542.459,E2 -4542.459} C_VEL
LIN {X 0,Y 530.93,Z 203.346,A -85,B 0,C 180,E1 -4543.611,E2 -4543.611} C_VEL
LIN {X 0,Y 530.259,Z 203.435,A -85,B 0,C 180,E1 -4544.245,E2 -4544.245} C_VEL
LIN {X 0,Y 527.409,Z 203.784,A -85,B 0,C 180,E1 -4545.273,E2 -4545.273} C_VEL
LIN {X 0,Y 525.004,Z 204.092,A -85,B 0,C 180,E1 -4546.102,E2 -4546.102} C_VEL
LIN {X 0,Y 523.973,Z 204.213,A -85,B 0,C 180,E1 -4546.742,E2 -4546.742} C_VEL
LIN {X 0,Y 523.889,Z 204.222,A -85,B 0,C 180,E1 -4546.958,E2 -4546.958} C_VEL
LIN {X 0,Y 523.953,Z 204.223,A -85,B 0,C 180,E1 -4549.926,E2 -4549.926} C_VEL
LIN {X 0,Y 523.889,Z 204.222,A -85,B 0,C 180,E1 -4552.871,E2 -4552.871} C_VEL
LIN {X 0,Y 523.926,Z 204.224,A -85,B 0,C 180,E1 -4555.714,E2 -4555.714} C_VEL
LIN {X 0,Y 523.916,Z 204.22,A -85,B 0,C 180,E1 -4558.46,E2 -4558.46} C_VEL
LIN {X 0,Y 523.929,Z 204.218,A -85,B 0,C 180,E1 -4561.128,E2 -4561.128} C_VEL
LIN {X 0,Y 523.974,Z 204.216,A -85,B 0,C 180,E1 -4563.982,E2 -4563.982} C_VEL
LIN {X 0,Y 523.926,Z 204.219,A -85,B 0,C 180,E1 -4566.273,E2 -4566.273} C_VEL
LIN {X 0,Y 523.937,Z 204.216,A -85,B 0,C 180,E1 -4568.769,E2 -4568.769} C_VEL
LIN {X 0,Y 523.944,Z 204.219,A -85,B 0,C 180,E1 -4571.223,E2 -4571.223} C_VEL
LIN {X 0,Y 523.932,Z 204.224,A -85,B 0,C 180,E1 -4573.641,E2 -4573.641} C_VEL
LIN {X 0,Y 523.94,Z 204.217,A -85,B 0,C 180,E1 -4576.03,E2 -4576.03} C_VEL
LIN {X 0,Y 524.009,Z 204.207,A -85,B 0,C 180,E1 -4578.395,E2 -4578.395} C_VEL
LIN {X 0,Y 524.002,Z 204.215,A -85,B 0,C 180,E1 -4581.517,E2 -4581.517} C_VEL
LIN {X 0,Y 524.08,Z 204.199,A -85,B 0,C 180,E1 -4584.614,E2 -4584.614} C_VEL
LIN {X 0,Y 524.112,Z 204.197,A -85,B 0,C 180,E1 -4587.695,E2 -4587.695} C_VEL
LIN {X 0,Y 524.121,Z 204.196,A -85,B 0,C 180,E1 -4590.768,E2 -4590.768} C_VEL
LIN {X 0,Y 524.07,Z 204.208,A -85,B 0,C 180,E1 -4593.075,E2 -4593.075} C_VEL
LIN {X 0,Y 524.032,Z 204.204,A -85,B 0,C 180,E1 -4596.159,E2 -4596.159} C_VEL
LIN {X 0,Y 524.002,Z 204.21,A -85,B 0,C 180,E1 -4598.483,E2 -4598.483} C_VEL
LIN {X 0,Y 524,Z 204.209,A -85,B 0,C 180,E1 -4601.738,E2 -4601.738} C_VEL
LIN {X 0,Y 523.988,Z 204.217,A -85,B 0,C 180,E1 -4605.051,E2 -4605.051} C_VEL
LIN {X 0,Y 523.958,Z 204.213,A -85,B 0,C 180,E1 -4607.967,E2 -4607.967} C_VEL
LIN {X 0,Y 523.965,Z 204.216,A -85,B 0,C 180,E1 -4610.408,E2 -4610.408} C_VEL
LIN {X 0,Y 523.908,Z 204.227,A -85,B 0,C 180,E1 -4612.891,E2 -4612.891} C_VEL
LIN {X 0,Y 523.944,Z 204.217,A -85,B 0,C 180,E1 -4615.416,E2 -4615.416} C_VEL
LIN {X 0,Y 523.958,Z 204.216,A -85,B 0,C 180,E1 -4617.996,E2 -4617.996} C_VEL
LIN {X 0,Y 524.043,Z 204.319,A -85,B 0,C 180,E1 -4621.068,E2 -4621.068} C_VEL
LIN {X 0,Y 524.416,Z 208.735,A -85,B 0,C 180,E1 -4621.952,E2 -4621.952} C_VEL
LIN {X 0,Y 524.232,Z 223.97,A -85,B 0,C 180,E1 -4624.914,E2 -4624.914} C_VEL
LIN {X 0,Y 525.955,Z 234.01,A -85,B 0,C 180,E1 -4625.109,E2 -4625.109} C_VEL
LIN {X 0,Y 525.449,Z 330.978,A -85,B 0,C 180,E1 -4626.475,E2 -4626.475} C_VEL
LIN {X 0,Y 525.258,Z 344.281,A -85,B 0,C 180,E1 -4626.823,E2 -4626.823} C_VEL
LIN {X 0,Y 525.107,Z 355.846,A -85,B 0,C 180,E1 -4627.269,E2 -4627.269} C_VEL
LIN {X 0,Y 524.88,Z 367.652,A -85,B 0,C 180,E1 -4627.878,E2 -4627.878} C_VEL
LIN {X 0,Y 524.578,Z 379.129,A -85,B 0,C 180,E1 -4628.643,E2 -4628.643} C_VEL
LIN {X 0,Y 524.305,Z 389.849,A -85,B 0,C 180,E1 -4629.542,E2 -4629.542} C_VEL
LIN {X 0,Y 524.048,Z 399.833,A -85,B 0,C 180,E1 -4630.588,E2 -4630.588} C_VEL
LIN {X 0,Y 523.839,Z 408.29,A -85,B 0,C 180,E1 -4631.687,E2 -4631.687} C_VEL
LIN {X 0,Y 523.622,Z 416.271,A -85,B 0,C 180,E1 -4632.986,E2 -4632.986} C_VEL
LIN {X 0,Y 523.532,Z 422.394,A -85,B 0,C 180,E1 -4634.265,E2 -4634.265} C_VEL
LIN {X 0,Y 523.423,Z 426.499,A -85,B 0,C 180,E1 -4635.361,E2 -4635.361} C_VEL
LIN {X 0,Y 523.367,Z 430.386,A -85,B 0,C 180,E1 -4636.777,E2 -4636.777} C_VEL
LIN {X 0,Y 523.334,Z 432.324,A -85,B 0,C 180,E1 -4637.82,E2 -4637.82} C_VEL
LIN {X 0,Y 523.33,Z 433.519,A -85,B 0,C 180,E1 -4638.85,E2 -4638.85} C_VEL
LIN {X 0,Y 523.262,Z 433.991,A -85,B 0,C 180,E1 -4639.951,E2 -4639.951} C_VEL
LIN {X 0,Y 523.281,Z 433.584,A -85,B 0,C 180,E1 -4641.159,E2 -4641.159} C_VEL
LIN {X 0,Y 523.288,Z 432.155,A -85,B 0,C 180,E1 -4642.402,E2 -4642.402} C_VEL
LIN {X 0,Y 523.407,Z 429.291,A -85,B 0,C 180,E1 -4643.786,E2 -4643.786} C_VEL
LIN {X 0,Y 523.416,Z 425.691,A -85,B 0,C 180,E1 -4644.982,E2 -4644.982} C_VEL
LIN {X 0,Y 523.546,Z 420.25,A -85,B 0,C 180,E1 -4646.324,E2 -4646.324} C_VEL
LIN {X 0,Y 523.687,Z 413.923,A -85,B 0,C 180,E1 -4647.534,E2 -4647.534} C_VEL
LIN {X 0,Y 523.869,Z 406.716,A -85,B 0,C 180,E1 -4648.638,E2 -4648.638} C_VEL
LIN {X 0,Y 524.146,Z 397.165,A -85,B 0,C 180,E1 -4649.814,E2 -4649.814} C_VEL
LIN {X 0,Y 524.383,Z 387.226,A -85,B 0,C 180,E1 -4650.796,E2 -4650.796} C_VEL
LIN {X 0,Y 524.603,Z 377.145,A -85,B 0,C 180,E1 -4651.603,E2 -4651.603} C_VEL
LIN {X 0,Y 524.902,Z 365.765,A -85,B 0,C 180,E1 -4652.327,E2 -4652.327} C_VEL
LIN {X 0,Y 525.163,Z 353.309,A -85,B 0,C 180,E1 -4652.935,E2 -4652.935} C_VEL
LIN {X 0,Y 525.36,Z 340.222,A -85,B 0,C 180,E1 -4653.393,E2 -4653.393} C_VEL
LIN {X 0,Y 525.508,Z 327.399,A -85,B 0,C 180,E1 -4653.678,E2 -4653.678} C_VEL
LIN {X 0,Y 525.928,Z 232.956,A -85,B 0,C 180,E1 -4655.001,E2 -4655.001} C_VEL
LIN {X 0,Y 524.188,Z 223.662,A -85,B 0,C 180,E1 -4655.204,E2 -4655.204} C_VEL
LIN {X 0,Y 524.204,Z 208.176,A -85,B 0,C 180,E1 -4657.952,E2 -4657.952} C_VEL
LIN {X 0,Y 523.972,Z 204.218,A -85,B 0,C 180,E1 -4658.665,E2 -4658.665} C_VEL
LIN {X 0,Y 523.909,Z 204.228,A -85,B 0,C 180,E1 -4661.219,E2 -4661.219} C_VEL
LIN {X 0,Y 523.907,Z 204.228,A -85,B 0,C 180,E1 -4663.638,E2 -4663.638} C_VEL
LIN {X 0,Y 523.899,Z 204.225,A -85,B 0,C 180,E1 -4666.027,E2 -4666.027} C_VEL
LIN {X 0,Y 523.965,Z 204.216,A -85,B 0,C 180,E1 -4668.393,E2 -4668.393} C_VEL
LIN {X 0,Y 523.956,Z 204.22,A -85,B 0,C 180,E1 -4671.515,E2 -4671.515} C_VEL
LIN {X 0,Y 523.998,Z 204.211,A -85,B 0,C 180,E1 -4673.841,E2 -4673.841} C_VEL
LIN {X 0,Y 524.025,Z 204.212,A -85,B 0,C 180,E1 -4676.925,E2 -4676.925} C_VEL
LIN {X 0,Y 524.052,Z 204.203,A -85,B 0,C 180,E1 -4680,E2 -4680} C_VEL
LIN {X 0,Y 524.023,Z 204.213,A -85,B 0,C 180,E1 -4683.075,E2 -4683.075} C_VEL
LIN {X 0,Y 523.982,Z 204.21,A -85,B 0,C 180,E1 -4686.16,E2 -4686.16} C_VEL
LIN {X 0,Y 523.952,Z 204.219,A -85,B 0,C 180,E1 -4689.263,E2 -4689.263} C_VEL
LIN {X 0,Y 523.972,Z 204.211,A -85,B 0,C 180,E1 -4691.753,E2 -4691.753} C_VEL
LIN {X 0,Y 523.94,Z 204.221,A -85,B 0,C 180,E1 -4695.054,E2 -4695.054} C_VEL
LIN {X 0,Y 523.921,Z 204.218,A -85,B 0,C 180,E1 -4697.971,E2 -4697.971} C_VEL
LIN {X 0,Y 523.925,Z 204.223,A -85,B 0,C 180,E1 -4700.412,E2 -4700.412} C_VEL
LIN {X 0,Y 523.896,Z 204.225,A -85,B 0,C 180,E1 -4702.895,E2 -4702.895} C_VEL
LIN {X 0,Y 523.941,Z 204.218,A -85,B 0,C 180,E1 -4706.023,E2 -4706.023} C_VEL
LIN {X 0,Y 523.9,Z 204.223,A -85,B 0,C 180,E1 -4708.877,E2 -4708.877} C_VEL
LIN {X 0,Y 523.891,Z 204.222,A -85,B 0,C 180,E1 -4711.546,E2 -4711.546} C_VEL
LIN {X 0,Y 523.905,Z 204.228,A -85,B 0,C 180,E1 -4714.293,E2 -4714.293} C_VEL
LIN {X 0,Y 523.878,Z 204.224,A -85,B 0,C 180,E1 -4717.135,E2 -4717.135} C_VEL
LIN {X 0,Y 523.906,Z 204.227,A -85,B 0,C 180,E1 -4720.133,E2 -4720.133} C_VEL
LIN {X 0,Y 523.908,Z 204.225,A -85,B 0,C 180,E1 -4722.462,E2 -4722.462} C_VEL
LIN {X 0,Y 523.918,Z 204.218,A -85,B 0,C 180,E1 -4725.313,E2 -4725.313} C_VEL
LIN {X 0,Y 523.938,Z 204.218,A -85,B 0,C 180,E1 -4728.692,E2 -4728.692} C_VEL
LIN {X 0,Y 523.896,Z 204.228,A -85,B 0,C 180,E1 -4731.901,E2 -4731.901} C_VEL
LIN {X 0,Y 523.919,Z 204.219,A -85,B 0,C 180,E1 -4734.913,E2 -4734.913} C_VEL
LIN {X 0,Y 523.921,Z 204.224,A -85,B 0,C 180,E1 -4737.683,E2 -4737.683} C_VEL
LIN {X 0,Y 523.943,Z 204.219,A -85,B 0,C 180,E1 -4740.679,E2 -4740.679} C_VEL
LIN {X 0,Y 523.964,Z 204.222,A -85,B 0,C 180,E1 -4743.731,E2 -4743.731} C_VEL
LIN {X 0,Y 524.01,Z 204.333,A -85,B 0,C 180,E1 -4745.276,E2 -4745.276} C_VEL
LIN {X 0,Y 525.273,Z 212.454,A -85,B 0,C 180,E1 -4746.547,E2 -4746.547} C_VEL
LIN {X 0,Y 524.919,Z 231.982,A -85,B 0,C 180,E1 -4749.447,E2 -4749.447} C_VEL
LIN {X 0,Y 524.517,Z 253.784,A -85,B 0,C 180,E1 -4752.657,E2 -4752.657} C_VEL
LIN {X 0,Y 524.255,Z 268.841,A -85,B 0,C 180,E1 -4754.843,E2 -4754.843} C_VEL
LIN {X 0,Y 525.885,Z 281.479,A -85,B 0,C 180,E1 -4755.07,E2 -4755.07} C_VEL
LIN {X 0,Y 525.443,Z 377.377,A -85,B 0,C 180,E1 -4756.415,E2 -4756.415} C_VEL
LIN {X 0,Y 525.233,Z 390.698,A -85,B 0,C 180,E1 -4756.755,E2 -4756.755} C_VEL
LIN {X 0,Y 524.94,Z 403.48,A -85,B 0,C 180,E1 -4757.239,E2 -4757.239} C_VEL
LIN {X 0,Y 524.769,Z 414.86,A -85,B 0,C 180,E1 -4757.824,E2 -4757.824} C_VEL
LIN {X 0,Y 524.433,Z 426.586,A -85,B 0,C 180,E1 -4758.601,E2 -4758.601} C_VEL
LIN {X 0,Y 524.179,Z 437.147,A -85,B 0,C 180,E1 -4759.475,E2 -4759.475} C_VEL
LIN {X 0,Y 523.955,Z 445.779,A -85,B 0,C 180,E1 -4760.349,E2 -4760.349} C_VEL
LIN {X 0,Y 523.757,Z 453.741,A -85,B 0,C 180,E1 -4761.318,E2 -4761.318} C_VEL
LIN {X 0,Y 523.578,Z 461.517,A -85,B 0,C 180,E1 -4762.481,E2 -4762.481} C_VEL
LIN {X 0,Y 523.467,Z 468.677,A -85,B 0,C 180,E1 -4763.835,E2 -4763.835} C_VEL
LIN {X 0,Y 523.383,Z 473.442,A -85,B 0,C 180,E1 -4764.993,E2 -4764.993} C_VEL
LIN {X 0,Y 523.443,Z 477.088,A -85,B 0,C 180,E1 -4766.151,E2 -4766.151} C_VEL
LIN {X 0,Y 523.367,Z 478.966,A -85,B 0,C 180,E1 -4766.921,E2 -4766.921} C_VEL
LIN {X 0,Y 523.335,Z 480.373,A -85,B 0,C 180,E1 -4767.691,E2 -4767.691} C_VEL
LIN {X 0,Y 523.258,Z 481.992,A -85,B 0,C 180,E1 -4769.23,E2 -4769.23} C_VEL
LIN {X 0,Y 523.259,Z 482.214,A -85,B 0,C 180,E1 -4770,E2 -4770} C_VEL
LIN {X 0,Y 523.275,Z 481.391,A -85,B 0,C 180,E1 -4771.539,E2 -4771.539} C_VEL
LIN {X 0,Y 523.335,Z 480.395,A -85,B 0,C 180,E1 -4772.309,E2 -4772.309} C_VEL
LIN {X 0,Y 523.367,Z 478.994,A -85,B 0,C 180,E1 -4773.079,E2 -4773.079} C_VEL
LIN {X 0,Y 523.423,Z 476.045,A -85,B 0,C 180,E1 -4774.235,E2 -4774.235} C_VEL
LIN {X 0,Y 523.456,Z 472.049,A -85,B 0,C 180,E1 -4775.392,E2 -4775.392} C_VEL
LIN {X 0,Y 523.508,Z 466.831,A -85,B 0,C 180,E1 -4776.566,E2 -4776.566} C_VEL
LIN {X 0,Y 523.613,Z 460.42,A -85,B 0,C 180,E1 -4777.713,E2 -4777.713} C_VEL
LIN {X 0,Y 523.801,Z 452.34,A -85,B 0,C 180,E1 -4778.875,E2 -4778.875} C_VEL
LIN {X 0,Y 523.984,Z 444.1,A -85,B 0,C 180,E1 -4779.845,E2 -4779.845} C_VEL
LIN {X 0,Y 524.3,Z 434.054,A -85,B 0,C 180,E1 -4780.815,E2 -4780.815} C_VEL
LIN {X 0,Y 524.549,Z 422.707,A -85,B 0,C 180,E1 -4781.689,E2 -4781.689} C_VEL
LIN {X 0,Y 524.821,Z 411.545,A -85,B 0,C 180,E1 -4782.371,E2 -4782.371} C_VEL
LIN {X 0,Y 525.07,Z 399.17,A -85,B 0,C 180,E1 -4782.954,E2 -4782.954} C_VEL
LIN {X 0,Y 525.327,Z 386.027,A -85,B 0,C 180,E1 -4783.39,E2 -4783.39} C_VEL
LIN {X 0,Y 525.481,Z 373.431,A -85,B 0,C 180,E1 -4783.657,E2 -4783.657} C_VEL
LIN {X 0,Y 525.814,Z 279.671,A -85,B 0,C 180,E1 -4784.961,E2 -4784.961} C_VEL
LIN {X 0,Y 524.285,Z 269.097,A -85,B 0,C 180,E1 -4785.169,E2 -4785.169} C_VEL
LIN {X 0,Y 524.688,Z 248.024,A -85,B 0,C 180,E1 -4788.305,E2 -4788.305} C_VEL
LIN {X 0,Y 525.206,Z 227.521,A -85,B 0,C 180,E1 -4791.383,E2 -4791.383} C_VEL
LIN {X 0,Y 525.557,Z 212.743,A -85,B 0,C 180,E1 -4793.649,E2 -4793.649} C_VEL
LIN {X 0,Y 524.003,Z 204.213,A -85,B 0,C 180,E1 -4795.068,E2 -4795.068} C_VEL
LIN {X 0,Y 523.953,Z 204.222,A -85,B 0,C 180,E1 -4797.996,E2 -4797.996} C_VEL
LIN {X 0,Y 523.931,Z 204.218,A -85,B 0,C 180,E1 -4800.852,E2 -4800.852} C_VEL
LIN {X 0,Y 523.945,Z 204.22,A -85,B 0,C 180,E1 -4803.731,E2 -4803.731} C_VEL
LIN {X 0,Y 523.902,Z 204.223,A -85,B 0,C 180,E1 -4806.401,E2 -4806.401} C_VEL
LIN {X 0,Y 523.9,Z 204.221,A -85,B 0,C 180,E1 -4809.081,E2 -4809.081} C_VEL
LIN {X 0,Y 523.932,Z 204.222,A -85,B 0,C 180,E1 -4812.115,E2 -4812.115} C_VEL
LIN {X 0,Y 523.927,Z 204.22,A -85,B 0,C 180,E1 -4815.305,E2 -4815.305} C_VEL
LIN {X 0,Y 523.93,Z 204.217,A -85,B 0,C 180,E1 -4818.686,E2 -4818.686} C_VEL
LIN {X 0,Y 523.881,Z 204.229,A -85,B 0,C 180,E1 -4821.895,E2 -4821.895} C_VEL
LIN {X 0,Y 523.902,Z 204.221,A -85,B 0,C 180,E1 -4824.906,E2 -4824.906} C_VEL
LIN {X 0,Y 523.903,Z 204.227,A -85,B 0,C 180,E1 -4827.675,E2 -4827.675} C_VEL
LIN {X 0,Y 523.913,Z 204.219,A -85,B 0,C 180,E1 -4830.673,E2 -4830.673} C_VEL
LIN {X 0,Y 523.932,Z 204.221,A -85,B 0,C 180,E1 -4833.726,E2 -4833.726} C_VEL
LIN {X 0,Y 523.902,Z 204.22,A -85,B 0,C 180,E1 -4836.269,E2 -4836.269} C_VEL
LIN {X 0,Y 523.904,Z 204.222,A -85,B 0,C 180,E1 -4838.765,E2 -4838.765} C_VEL
LIN {X 0,Y 523.907,Z 204.228,A -85,B 0,C 180,E1 -4841.219,E2 -4841.219} C_VEL
LIN {X 0,Y 523.904,Z 204.224,A -85,B 0,C 180,E1 -4843.638,E2 -4843.638} C_VEL
LIN {X 0,Y 523.886,Z 204.223,A -85,B 0,C 180,E1 -4846.026,E2 -4846.026} C_VEL
LIN {X 0,Y 523.964,Z 204.221,A -85,B 0,C 180,E1 -4849.176,E2 -4849.176} C_VEL
LIN {X 0,Y 523.973,Z 204.212,A -85,B 0,C 180,E1 -4852.291,E2 -4852.291} C_VEL
